///////////////////////////////////////////////////////////////////////////////////////////////////////////////////
	ELSIF StartAction('Nom Action') THEN
		CASE G_Match.iEtapeAction OF
			0:
				IF "CONDITION POUR L'ETAPE SUIVANTE" THEN
					Next(); //etape suivante
				END_IF
			1:
				IF "FIN DE L'ACTION" THEN
					FinishAction(0,0);
				END_IF
		END_CASE
____________________________________________________________________________________________________________________

-> CASE POUR UNE ACTION ASYNCHRONE AVEC LE TABLEAU 
continue la suite du Tableau et l'action en même temps. Si le tableau arrive à une autre action, 
l'action asynchrone est terminée avant de commencer la prochaine action

///////////////////////////////////////////////////////////////////////////////////////////////////////////////////
	ELSIF StartAction('Nom Action') THEN
		CASE G_Match.iEtapeAction OF
			0:
				G_Match.iEtapeAction := G_Match.iEtapeAction + 1;
			1:
				FinishAction(StartAsync := TRUE,0);
			2:
				FinishAction(0,StopAsync := TRUE);
		END_CASE
____________________________________________________________________________________________________________________
*)
END_ACTION

ACTION _5_Interruption_active:
ITMotion.odometrie.M_reset_moteurs();

//Si le robot est bloqué depuis trop longtemps, il essaye différentes actions
IF IbAbortTask THEN
	//Check si c'est possible de reculer en attendant
	(*
	G_Odometrie.lrPositionX;
	G_Odometrie.lrPositionY;
	G_Match.Tableau[G_Match.iLigne].lrPositionX_mm;
	G_Match.Tableau[G_Match.iLigne].lrPositionY_mm;
	G_Balise.lrCoord_X1;
	G_Balise.lrCoord_Y1;
	G_Balise.lrDistance_1;
	*)

	//Sinon calcule les points de la mission en cours
	
	//Vérifie les stratégie possible selon la position
	
	//Choisi la meilleur stratégie à adopter
	
	//modifie le tableau
	
	pass();
END_IF

(*
Adaptation de la stratégie:
- Calcul des points restants
- Recherche de la prochaine stratégie
- Adaptation potentiel du programme
- Changement d'étape et déduction de points
*)

(*
- Tourner 90 degré
- move curve
- reprise de trajectoire

if coordX < 0 or coordX > 3000 or coordY > 2000 or coordY < 0 then
*)
END_ACTION

ACTION _6_Timeout_active:
//S'il ne reste plus de temps pour le match, le robot entamme la manoeuvre pour rentrer à la base
tempTableau.TypeTache := eChangementTache;
tempTableau.EtapeCible := 'retour base';
ReplaceStep(tempTableau);
G_Match.RetourEnCours := TRUE;
END_ACTION

ACTION _7_EndMatch_active:

VisuElems.CURRENTVISU 	:= 'V_Fin_Match';

//arrêt de tous les mouvements
IF G_Match.MatchEnCours THEN
	FOR G_EndMatch.icounter := 1 TO IiNumDynamixel DO
		ITAction.DXLIN[G_EndMatch.icounter].bGetLoad 		:= FALSE;
		ITAction.DXLIN[G_EndMatch.icounter].bGetMovement 	:= FALSE;
		ITAction.DXLIN[G_EndMatch.icounter].bGetPosition 	:= FALSE;

		ITAction.DXLIN[G_EndMatch.icounter].ParamReset_BOOL := TRUE;
		ITAction.DXLIN[G_EndMatch.icounter].bStopPosition 	:= TRUE;
	END_FOR
	
	QbMoteurStop 			:= TRUE;
	G_Match.MatchEnCours 	:= FALSE;
	G_Match.RetourEnCours	:= FALSE;
	baseTime := TIME();
END_IF

//attente pour être sûr que tout soit bien arrêté
IF delay(baseTime, T#0.5S)THEN
	QbMoteurStop 			:= FALSE;
	QbstartBalise 			:= FALSE;
	QbmoteurPower 			:= FALSE;
	
	FOR G_EndMatch.icounter := 1 TO IiNumDynamixel DO
		IF ITAction.DXLOUT[G_EndMatch.icounter].bStopPosition THEN 
			ITAction.DXLIN[G_EndMatch.icounter].bStopPosition := FALSE;
		END_IF
	END_FOR
	
	IF NOT IbStartMatch THEN
			G_EndMatch.bShutdown_done := TRUE;
	END_IF
END_IF;
END_ACTION

ACTION _Config_Visu_active:
IF G_Visus.bConfigEnable THEN 
	VisuElems.CURRENTVISU := 'V_Config';
	//Move robot
	ITMotion.odometrie.M_move_to_coordonne(
	x 			:= G_Visus.lrConfigPosX,
	y 			:= G_Visus.lrConfigPosY,
	lrSpeed 	:= G_Visus.lrConfigVitesse,
	bExecute 	:= G_Visus.bConfigStart,
	bbackward	:= G_Visus.bConfigMarcheArriere,
	bDone 		=> G_Visus.bConfigMoveDone);
	
	//set acceleration / deceleration
	IF G_Visus.lrConfigAcc <> 0 OR G_Visus.lrConfigDecc <> 0 THEN
		ITMotion.odometrie.M_set_acceleration(lrAcc := G_Visus.lrConfigAcc, lrDecc := G_Visus.lrConfigDecc);
	END_IF
	
	//balise on
	QbstartBalise := G_Visus.bConfigBalise;
	
	//moteur on
	QbmoteurPower := G_Visus.bConfigMoteurPower;
	
	//bouton reset
	IF G_Visus.bConfigReset THEN 
		ITMotion.odometrie.M_init_coordonne(bChoixCote := G_Visus.bConfigChoixCote);
	END_IF
	
	//erreur et pourcentage 
	G_Visus.lrConfigErreurX := ABS(G_odometrie.lrPositionX - G_Visus.lrConfigPosX);
	G_Visus.lrConfigErreurY := ABS(G_odometrie.lrPositionY - G_Visus.lrConfigPosY);
	G_Visus.lrConfigErreurX_Pourcent := ABS(G_Visus.lrConfigErreurX/G_odometrie.lrPositionX)*100;
	G_Visus.lrConfigErreurY_Pourcent := ABS(G_Visus.lrConfigErreurY/G_odometrie.lrPositionY)*100;

ELSE// désactivation du mode config
	
	//remise à 0 des valeurs
	QbstartBalise := FALSE;	
	QbmoteurPower := FALSE;
	G_Visus.lrConfigErreurX :=0 ;
	G_Visus.lrConfigErreurY := 0;
	G_Visus.lrConfigErreurX_Pourcent := 0;
	G_Visus.lrConfigErreurY_Pourcent := 0;
	G_Visus.bConfigStart := 0;
	
	//retour au menu
	VisuElems.CURRENTVISU := 'V_Menu';
END_IF

//On doit refaire un init après être sorti du mode config
G_init.binitDone := FALSE;

//mouvement prêt à être effectué
G_Visus.bConfigMoteurReady := IbMoteurOn;

//Indicateur pour dire que le robot est prêt à effectuer un déplacement
IF G_Visus.bConfigMoveDone THEN 
	G_Visus.bConfigStart := FALSE;
END_IF

IF G_Visus.bConfigMoteurReady AND (G_Visus.bConfigStart AND G_Visus.bConfigMoveDone OR NOT G_Visus.bConfigStart)THEN 
	G_Visus.bConfigReady := TRUE;
ELSE
	G_Visus.bConfigReady := FALSE;	
END_IF
END_ACTION

ACTION _Test_Visu_active:
//quitte le mode visu si on retourne au menu
IF VisuElems.CURRENTVISU = 'V_Test' THEN
	G_Visus.bTestEnable := TRUE;
ELSE
	G_Visus.bTestEnable := FALSE;
END_IF

//On doit refaire un init après être sorti du mode Test
G_init.binitDone := FALSE;

IF G_Visus.bTestEnable THEN 
	IF    G_Visus.sTestBouton1 THEN
		G_Match.Tableau[G_Match.iLigne].TypeAction := G_Visus.sTestFunction1;
	ELSIF G_Visus.sTestBouton2 THEN
		G_Match.Tableau[G_Match.iLigne].TypeAction := G_Visus.sTestFunction2;
	ELSIF G_Visus.sTestBouton3 THEN
		G_Match.Tableau[G_Match.iLigne].TypeAction := G_Visus.sTestFunction3;
	ELSIF G_Visus.sTestBouton4 THEN
		G_Match.Tableau[G_Match.iLigne].TypeAction := G_Visus.sTestFunction4;
	ELSIF G_Visus.sTestBouton5 THEN
		G_Match.Tableau[G_Match.iLigne].TypeAction := G_Visus.sTestFunction5;
	ELSIF G_Visus.sTestBouton6 THEN
		G_Match.Tableau[G_Match.iLigne].TypeAction := G_Visus.sTestFunction6;
	END_IF
	
	// TO DO !!!
	//Définir le nom des actions testées 
	G_Visus.sTestFunction1 := 'Dynamixel position 4095';
	G_Visus.sTestFunction2 := 'Dynamixel position 0';
	G_Visus.sTestFunction3 := 'None';
	G_Visus.sTestFunction4 := 'None';
	G_Visus.sTestFunction5 := 'None';
	G_Visus.sTestFunction6 := 'None';
	
	///////////////////////////////////////////////////////////////////////////////////////////////////////////////////
	// GESTION DES ACTIONS 
	///////////////////////////////////////////////////////////////////////////////////////////////////////////////////
	IF StartAction('Dynamixel position 4095') THEN
		CASE G_Match.iEtapeAction OF
			0:
				ITAction.DXLIN[ITAction.MoteurXL1].bPosition := TRUE;
				ITAction.DXLIN[ITAction.MoteurXL1].ParamPosition_DINT := 4095;
				ITAction.DXLIN[ITAction.MoteurXL1].ParamSpeed_INT := 500;
				IF ITAction.DXLOUT[ITAction.MoteurXL1].bPosition THEN
					ITAction.DXLIN[ITAction.MoteurXL1].bPosition := FALSE;
					Next();
				END_IF
			1:
				ITAction.DXLIN[ITAction.MoteurXL1].bGetPosition := TRUE;
				IF PlusOuMoins(ITAction.DXLOUT[ITAction.MoteurXL1].INFO_Position_dint, 4095, 15) THEN 
					ITAction.DXLIN[ITAction.MoteurXL1].bGetPosition := FALSE;
					FinishAction(0);
				END_IF
		END_CASE
	//__________________________________________________________________________________________________________________
	///////////////////////////////////////////////////////////////////////////////////////////////////////////////////			
	ELSIF StartAction('Dynamixel position 0') THEN
		CASE G_Match.iEtapeAction OF
			0:
				ITAction.DXLIN[ITAction.MoteurXL1].bPosition := TRUE;
				ITAction.DXLIN[ITAction.MoteurXL1].ParamPosition_DINT := 1;
				ITAction.DXLIN[ITAction.MoteurXL1].ParamSpeed_INT := 1030;
				IF ITAction.DXLOUT[ITAction.MoteurXL1].bPosition THEN
					ITAction.DXLIN[ITAction.MoteurXL1].bPosition := FALSE;
					Next();;
				END_IF
			1:
				ITAction.DXLIN[ITAction.MoteurXL1].bGetPosition := TRUE;
				IF PlusOuMoins(ITAction.DXLOUT[ITAction.MoteurXL1].INFO_Position_dint, 1, 15) THEN 
					ITAction.DXLIN[ITAction.MoteurXL1].bGetPosition := FALSE;
					FinishAction(0);
				END_IF
		END_CASE
	//__________________________________________________________________________________________________________________
	///////////////////////////////////////////////////////////////////////////////////////////////////////////////////	
	END_IF
	
	//Action terminée
	if G_Match.bActionFinie then
		G_Match.Tableau[G_Match.iLigne].TypeAction := '';
		G_Match.bActionFinie := FALSE;
		G_Match.iEtapeAction := 0;
		
		G_Visus.sTestBouton1 := FALSE;
		G_Visus.sTestBouton2 := FALSE;
		G_Visus.sTestBouton3 := FALSE;
		G_Visus.sTestBouton4 := FALSE;
		G_Visus.sTestBouton5 := FALSE;
		G_Visus.sTestBouton6 := FALSE;
	END_IF

ELSE// désactivation du mode Test
	//remise à 0 des valeurs
	G_Match.bActionFinie := FALSE;
	G_Match.Tableau[G_Match.iLigne].TypeAction := '';
	G_Match.iEtapeAction := 0;
	
	G_Visus.sTestBouton1 := FALSE;
	G_Visus.sTestBouton2 := FALSE;
	G_Visus.sTestBouton3 := FALSE;
	G_Visus.sTestBouton4 := FALSE;
	G_Visus.sTestBouton5 := FALSE;
	G_Visus.sTestBouton6 := FALSE;
	
	FOR G_Match.icounter := 1 TO IiNumDynamixel DO
		ITAction.DXLIN[G_Match.icounter].bGetLoad 		:= FALSE;
		ITAction.DXLIN[G_Match.icounter].bGetMovement 	:= FALSE;
		ITAction.DXLIN[G_Match.icounter].bGetPosition 	:= FALSE;
	END_FOR
END_IF
END_ACTION

TRANSITION T_ArreteTout:
IbEndMatch or G_Match.TimeMatch >= T#100s
END_TRANSITION

TRANSITION T_finMatchNormal:
G_Match.Tableau[G_Match.iLigne].TypeTache = eFinParcours;
END_TRANSITION

TRANSITION T_RetourMatch:
NOT IbPauseMotion
END_TRANSITION

TRANSITION T_Timeout:
G_Match.TimeMatch > T#20s and not G_Match.RetourEnCours
END_TRANSITION

END_PROGRAM

// ---- POUs/Action/ITAction.TcPOU
PROGRAM ITAction
(*IMPORTANT !!! à modifier correctment selon les besoins*)
VAR CONSTANT
	//nombre total de dynamixel
	iNombreDynamixel 	: INT := 4;
	iNombreXL			: INT := 2;
	iNombreAX			: INT := 2;
	
	//définition de l'ID des dynamixels, tous les ID doivent se suivrent => ex: moteur_1 := 1,moteur_2 := 2, moteur_3 := 3, etc...
	//Si des moteurs AX-12A sont présents, leur ID doivent aller après celles des moteurs XL430 ou XL330 => ex: XL430_moteur_5 := 5, AX12A_moteur_1 := 6, etc...
	MoteurXL1 			: INT := 1; //exemple XL430
	MoteurXL2			: INT := 2;
	MoteurAX1 			: INT := 3; //exemple AX12A
	MoteurAX2			: INT := 4;
END_VAR	

VAR_INPUT
	//démarrage et arrêt du script python
	IbStartPyscript 	: BOOL;
	IbStopPyscript		: BOOL;

	//envoi de commande aux moteurs Dynamixel
	DXLIN 				: ARRAY [1..iNombreDynamixel] OF ST_Dynamixel_Control_Input;
END_VAR

VAR_OUTPUT
	QbPyScriptRunning 	: BOOL; //le script python est actif
	QiNombreDynamixel	: INT;
	//retour d'informations des moteurs Dynamixel
	DXLOUT 				: ARRAY [1..iNombreDynamixel] OF ST_Dynamixel_Control_Output;
END_VAR

QiNombreDynamixel := iNombreDynamixel;
P_DXL_launch_pyscript(bstart := IbStartPyscript, bstop := IbStopPyscript);
QbPyScriptRunning := P_DXL_launch_pyscript.bActive;
P_connect_DXL(DXL_IN := DXLIN, DXL_OUT := DXLOUT);

END_PROGRAM

// ---- POUs/Action/Dynamixel/P_DXL_launch_pyscript.TcPOU
PROGRAM P_DXL_launch_pyscript
VAR_INPUT 
	bstart : BOOL;
	bstop : BOOL;
END_VAR
VAR_OUTPUT
	bActive : BOOL;
END_VAR
VAR
	start_python		:NT_StartProcess;
	get_AMSNETID		:FB_GetLocalAmsNetId;
	sPath 				:STRING:= '/C Python Dev\DXL_LIB\';
	sPython_script 		:STRING:= 'DXL_PYADS_PORT.py';
	sAMSNETID 			:STRING;	
	sLaunchCommandLine 	:STRING;
	bBusy				:BOOL;
	
	bRestart_active : BOOL;
END_VAR

//AMSnetID de l'automate
get_AMSNETID(bExecute:=TRUE,AddrString=>sAMSNETID, bBusy=>bBusy);

//ligne de commande dans le terminal pour lancer le script python
sLaunchCommandLine := CONCAT(sPath, sPython_script);
sLaunchCommandLine := CONCAT(sLaunchCommandLine, ' -a ');
sLaunchCommandLine := CONCAT(sLaunchCommandLine, sAMSNETID);

//lance une commande dans le terminal windows pour lancer le script python
//la commande est lancée depuis C:\Windows\SysWOW64\
IF NOT bBusy THEN
	start_python(
	NETID:= '',
	PATHSTR:= 'C:\Windows\System32\cmd.exe',
	DIRNAME:= '',
	COMNDLINE:= sLaunchCommandLine,
	START:= G_DXL.bRestart_py_script,
	TMOUT := T#5S,
	Busy=>,
	ERR=> ,
	ERRID=>); 
END_IF


IF bstart OR bRestart_active THEN 
	// active le script python 1 fois (done_internal bloque la réactivation une fois qu'il a été effectué)
	IF NOT G_DXL.bRestart_py_script AND NOT bRestart_active THEN
		G_DXL.bRestart_py_script := TRUE;
		bRestart_active := TRUE;
	END_IF
	
	// désactive le script python si il était activé
	IF G_DXL.bRestart_py_script AND NOT G_DXL.bPyscript_running AND NOT bRestart_active THEN
		G_DXL.bRestart_py_script := FALSE;	
	END_IF
	
	// libére la réactivation du script python lorsqu'il à redémarré
	IF bRestart_active AND G_DXL.bPyscript_running THEN
		bRestart_active := FALSE;
	END_IF
END_IF

//arrête le script python
IF bStop THEN 
	G_DXL.bStop_python_script := TRUE;
ELSE
	G_DXL.bStop_python_script := FALSE;
END_IF

bActive := G_DXL.bPyscript_running;

END_PROGRAM

// ---- POUs/Action/Dynamixel/P_Connect_DXL.TcPOU
PROGRAM P_Connect_DXL
VAR_IN_OUT
	DXL_IN 	: ARRAY [1..ITAction.iNombreDynamixel] OF ST_Dynamixel_Control_Input;
	DXL_OUT : ARRAY [1..ITAction.iNombreDynamixel] OF ST_Dynamixel_Control_Output;
END_VAR
VAR
	icounter : INT;
END_VAR

FOR icounter := 1 TO ITAction.iNombreDynamixel DO
	IF icounter <= ITAction.iNombreXL THEN //Définition des moteurs XL430 et XL330
		DXL_IN[icounter].TypeXL							(id:= icounter);
		DXL_IN[icounter].TypeXL.send_enable_torque		(EN:=DXL_IN[icounter].bEnableTorque, 	done=> DXL_OUT[icounter].bEnableTorque);
		DXL_IN[icounter].TypeXL.send_disable_torque		(EN:=DXL_IN[icounter].bDisableTorque, 	done=> DXL_OUT[icounter].bDisableTorque);
		DXL_IN[icounter].TypeXL.send_led_on				(EN:=DXL_IN[icounter].bLedOn, 			done=> DXL_OUT[icounter].bLedOn);		
		DXL_IN[icounter].TypeXL.send_led_off			(EN:=DXL_IN[icounter].IbLedOff, 		done=> DXL_OUT[icounter].bLedOff);
		DXL_IN[icounter].TypeXL.send_operating_mode		(EN:=DXL_IN[icounter].bOperatingMode,	done=> DXL_OUT[icounter].bOperatingMode,mode:= DXL_IN[icounter].ParamOperatingMode_string);
		DXL_IN[icounter].TypeXL.send_position			(EN:=DXL_IN[icounter].bPosition, 		done=> DXL_OUT[icounter].bPosition, position 	:= DXL_IN[icounter].ParamPosition_DINT, vitesse:= DXL_IN[icounter].ParamSpeed_INT);
		DXL_IN[icounter].TypeXL.send_stop_position		(EN:=DXL_IN[icounter].bStopPosition, 	done=> DXL_OUT[icounter].bStopPosition,reset:= DXL_IN[icounter].ParamReset_BOOL);
		DXL_IN[icounter].TypeXL.send_reset_position		(EN:=DXL_IN[icounter].bResetPosition, 	done=> DXL_OUT[icounter].bResetPosition);
		DXL_IN[icounter].TypeXL.send_acceleration		(EN:=DXL_IN[icounter].bAcceleration,	done=> DXL_OUT[icounter].bAcceleration, acceleration:= DXL_IN[icounter].ParamAcceleration_USINT, speed:=DXL_IN[icounter].ParamSpeed_INT);
		DXL_IN[icounter].TypeXL.send_velocity			(EN:=DXL_IN[icounter].bVelocity, 		done=> DXL_OUT[icounter].bVelocity, vitesse := DXL_IN[icounter].ParamSpeed_INT);
	    DXL_IN[icounter].TypeXL.get_load				(EN:=DXL_IN[icounter].bGetLoad, 		load=> DXL_OUT[icounter].INFO_load_int);
		DXL_IN[icounter].TypeXL.get_movement			(EN:=DXL_IN[icounter].bGetMovement, 	mouvement=> DXL_OUT[icounter].INFO_Mouvement_bool);
		DXL_IN[icounter].TypeXL.get_position			(EN:=DXL_IN[icounter].bGetPosition,	position=> DXL_OUT[icounter].INFO_Position_dint);
	ELSIF icounter > ITAction.iNombreAX THEN //définition des moteurs AX-12A
		DXL_IN[icounter].TypeAX							(id:= icounter);
		DXL_IN[icounter].TypeAX.send_enable_torque		(EN:=DXL_IN[icounter].bEnableTorque, 	done=> DXL_OUT[icounter].bEnableTorque);
		DXL_IN[icounter].TypeAX.send_disable_torque		(EN:=DXL_IN[icounter].bDisableTorque, 	done=> DXL_OUT[icounter].bDisableTorque);
		DXL_IN[icounter].TypeAX.send_led_on				(EN:=DXL_IN[icounter].bLedOn, 			done=> DXL_OUT[icounter].bLedOn);		
		DXL_IN[icounter].TypeAX.send_led_off			(EN:=DXL_IN[icounter].IbLedOff, 		done=> DXL_OUT[icounter].bLedOff);
		DXL_IN[icounter].TypeAX.send_operating_mode		(EN:=DXL_IN[icounter].bOperatingMode,	done=> DXL_OUT[icounter].bOperatingMode, mode:=DXL_IN[icounter].ParamOperatingMode_string, );
		DXL_IN[icounter].TypeAX.send_position			(EN:=DXL_IN[icounter].bPosition, 		done=> DXL_OUT[icounter].bPosition, position := DXL_IN[icounter].ParamPosition_DINT, vitesse:=DXL_IN[icounter].ParamSpeed_INT);
		DXL_IN[icounter].TypeAX.send_stop_position		(EN:=DXL_IN[icounter].bStopPosition, 	done=> DXL_OUT[icounter].bStopPosition);
		DXL_IN[icounter].TypeAX.send_velocity			(EN:=DXL_IN[icounter].bVelocity, 		done=> DXL_OUT[icounter].bVelocity, vitesse := DXL_IN[icounter].ParamSpeed_INT);
		DXL_IN[icounter].TypeAX.get_load				(EN:=DXL_IN[icounter].bGetLoad, 		load=> DXL_OUT[icounter].INFO_load_int);
		DXL_IN[icounter].TypeAX.get_movement			(EN:=DXL_IN[icounter].bGetMovement, 	mouvement=> DXL_OUT[icounter].INFO_Mouvement_bool);
		DXL_IN[icounter].TypeAX.get_position			(EN:=DXL_IN[icounter].bGetPosition,	position=> DXL_OUT[icounter].INFO_Position_dint);
	END_IF
END_FOR

END_PROGRAM

// ---- POUs/Utillity/Structure/Action/FinishAction.TcPOU
FUNCTION FinishAction 
VAR_INPUT
	StartAsync : BOOL := FALSE;
END_VAR
VAR
END_VAR

G_Match.bActionFinie := TRUE; //arrête l'action sans arrêter la partie asynchrone
IF NOT StartAsync THEN        //arrête l'action asynchrone
	G_Match.iAsyncAction := ''; 
	G_Match.iEtapeAction := 0;
END_IF

END_FUNCTION

// ---- POUs/Structure/Actions/F_DXL_Position.TcPOU
FUNCTION F_DXL_Position : bool
VAR_INPUT
	position:DINT;
	speed	:INT;
	ID		:INT;
END_VAR

CASE G_Match.iEtapeAction OF
	0:
		ITAction.DXLIN[ID].bPosition := TRUE;
		ITAction.DXLIN[ID].ParamPosition_DINT := position;
		ITAction.DXLIN[ID].ParamSpeed_INT := speed;
		IF ITAction.DXLOUT[ID].bPosition THEN
			ITAction.DXLIN[ID].bPosition := FALSE;
			FinishAction(1);
			Next();;
		END_IF
	1:
		ITAction.DXLIN[ID].bGetPosition := TRUE;
		IF PlusOuMoins(ITAction.DXLOUT[ID].INFO_Position_dint, 0, 15) THEN 
			ITAction.DXLIN[ITAction.MoteurXL1].bGetPosition := FALSE;
			FinishAction(0);
		END_IF
END_CASE

END_FUNCTION

// ---- POUs/Structure/Actions/F_DXL_Reset.TcPOU
FUNCTION F_DXL_Reset : bool
VAR_INPUT
	ID:INT;
	offset:DINT;
	
END_VAR
VAR_IN_OUT
	baseTime:TIME;
END_VAR
VAR
END_VAR

CASE G_Match.iEtapeAction OF
	0:
		ITAction.DXLIN[ID].ParamPosition_DINT := 100000;
		ITAction.DXLIN[ID].ParamSpeed_INT := 100;
		
		ITAction.DXLIN[ID].bPosition := TRUE;
		IF ITAction.DXLOUT[ID].bPosition THEN
			ITAction.DXLIN[ID].bPosition := FALSE;
			baseTime := TIME();
			Next();
		END_IF
	1:
		IF delay(baseTime,T#1S)THEN
			next();
		END_IF;
	2:
		G_Visus.bMatchEnemi := TRUE;
		ITAction.DXLIN[ID].bGetLoad := TRUE;
		IF  G_IO.bCaptDepart OR ITAction.DXLOUT[ID].INFO_load_int >= 150 THEN
			ITAction.DXLIN[ITAction.MoteurXL2].bGetLoad := FALSE;
			next();
		END_IF
	3:
		G_Visus.bMatchEnemi := FALSE;
		ITAction.DXLIN[ID].ParamReset_BOOL := TRUE;
		ITAction.DXLIN[ID].bStopPosition := TRUE;
		IF ITAction.DXLOUT[ID].bStopPosition THEN 
			ITAction.DXLIN[ID].bStopPosition := FALSE;
			next();
		END_IF
	4:
		ITAction.DXLIN[ID].bPosition := TRUE;
		ITAction.DXLIN[ID].ParamPosition_DINT := offset;
		ITAction.DXLIN[ID].ParamSpeed_INT := 500;
		IF ITAction.DXLOUT[ID].bPosition THEN
			ITAction.DXLIN[ID].bPosition := FALSE;
			FinishAction(0);
		END_IF
END_CASE

END_FUNCTION

// ---- POUs/Utillity/Structure/Tableau/ReplaceStep.TcPOU
FUNCTION ReplaceStep : bool
VAR_INPUT
	step:ST_Tableau;
END_VAR
VAR
END_VAR

//change l'étape actuelle
G_Match.Tableau[G_Match.iLigne] := step;

END_FUNCTION

// ---- POUs/Communication/ITCommunication.TcPOU
PROGRAM ITCommunication
VAR_INPUT
	IbStartConnection:BOOL;
	IbPublishStart:BOOL;
END_VAR
VAR_OUTPUT
	QbOnline : BOOL;
END_VAR
VAR
	//Lit l'adresse IP de l'automate
	FB_MDP_NIC_Read    : FB_MDP_NIC_Read;
	iAddPoint		   : INT;
END_VAR

FB_MDP_NIC_Read(bExecute := True, tTimeout := DEFAULT_ADS_TIMEOUT);
MQTT(IsHostIP := FB_MDP_NIC_Read.stMDP_ModuleContent.sIPAddress, IbConnect := IbStartConnection, IsTopicOut := 'StartPamis', IsTopicIn := 'FinParcours', IbPublishStart := IbPublishStart, IsPayload := 'Start', QiAddPoint := iAddPoint);
QbOnline := MQTT.QbOnline;

END_PROGRAM

// ---- POUs/Communication/MQTT.TcPOU
PROGRAM MQTT
VAR_INPUT
	IsHostIP 	: STRING;					//Adresse IP du broker Mosquitto qui tourne sur la partie windows de la PLC
	IbConnect 	: BOOL;						//Commence la connection MQTT
	
	IsTopicOut 	: STRING;					//Nom du Topic où la PLC publie des chose
	IsTopicIn 	: STRING;					//Nom du Topic où la PLC est souscrite (lis les informations)
	IbPublishStart : BOOL;					//Un front montant publie le message IsPayload dans le topic IsTopicOut
	IsPayload : STRING;						//Message à publier dans le topic
	
END_VAR
VAR_OUTPUT
	QbOnline : BOOL;						//Communication MQTT en ligne
END_VAR
VAR_IN_OUT
	QiAddPoint : INT;						//Donne l'ordre d'ajouter des points	
END_VAR
VAR
fbMqttClient 	: FB_IotMqttClient;			//FB de gestion de la communication MQTT
fbMessageQueue 	: FB_IotMqttMessageQueue;	//Zone tampon de stockage des messages reçus
fbMessage 		: FB_IotMqttMessage;		//Formattage des message MQTT reçu

RT_Publish 		: R_TRIG;					//Front montant pour la publication

bSubscribed : BOOL;							//Souscription au topic effectué

{attribute 'TcEncoding':='UTF-8'}
sPayloadRcv 	: STRING(255);				//Contenu du message souscrit (valeur reçue)
iNumPamiDone	: INT;						//Numéro du PAMI qui à fini son action
END_VAR

IF _TaskInfo[GETCURTASKINDEXEX()].FirstCycle THEN	//Lancement de la recherche de broker
	fbMqttClient.sHostName 		:= IsHostIP;		//Adresse IP d'ou se situe le broker (donc sur un Raspberry dans Node-red)
	fbMqttClient.nHostPort 		:= 1883;			//Port de communication du broker
	fbMqttClient.sClientId 		:= 'Bobst PLC';
	fbMqttClient.sTopicPrefix 	:= '';
	fbMqttClient.nKeepAlive 	:= 10;
	fbMqttClient.ipMessageQueue := fbMessageQueue;	//Sert à stocker les messages souscrit avant de les traiter
END_IF

//Lancement de la connexion MQTT
fbMqttClient.Execute(IbConnect);	
QbOnline := fbMqttClient.bConnected AND bSubscribed;

//Si on est connecté au broker alors...
IF fbMqttClient.bConnected THEN	

	//*** Souscrire à un topic ***//
	IF NOT bSubscribed THEN		//Signal pour lancer la souscription à un message
		bSubscribed := fbMqttClient.Subscribe(sTopic:=IsTopicIn,  eQoS:=TcIotMqttQos.AtMostOnceDelivery);
	END_IF
	
	//*** Publier un message ***//
	RT_Publish(clk:=IbPublishStart);
	IF  RT_Publish.Q THEN //Lorsque ce signal est à 1, on publie un message
		fbMqttClient.Publish( sTopic  		:= IsTopicOut,	//On écrit le nom du Topic d'un message à envoyer
							  pPayload		:= ADR(IsPayload),	//On écrit le contenu du message à envoyer (valeur à envoyer)
							  nPayloadSize	:= SIZEOF(IsPayload),	//On indique la taille du STRING donc le nombre de caractère.
							  eQoS			:= TcIotMqttQos.AtMostOnceDelivery,	//Qualité de service, à laisser comme cela
							  bRetain		:= FALSE,	//à laisser comme cela
							  bQueue		:= FALSE );	//à laisser comme cela
	END_IF			
END_IF

//*** Récupérer les messages des topics auquels on est souscris ***//
IF (fbMessageQueue.nQueuedMessages > 0) THEN 
	IF fbMessageQueue.Dequeue(fbMessage:=fbMessage) THEN
		IF fbMessage.CompareTopic(sTopic:=IsTopicIn) THEN
			fbMessage.GetPayload(pPayload:=ADR(sPayloadRcv), nPayloadSize:=SIZEOF(sPayloadRcv), bSetNullTermination:=FALSE);	//Valeur du message 1 reçu
		END_IF
		iNumPamiDone := STRING_TO_INT(RIGHT(sPayloadRcv,1));		
	END_IF
END_IF

//Choisi le nombre de points à ajouter en fonction du message MQTT reçu
CASE iNumPamiDone OF
	0:
		pass();
	1:
		QiAddPoint := 10;
		iNumPamiDone := 0;
	2:
		QiAddPoint := 10;
		iNumPamiDone := 0;
	3:
		QiAddPoint := 10;
		iNumPamiDone := 0;
	4:		
		QiAddPoint := 10;
		iNumPamiDone := 0;
END_CASE

END_PROGRAM

// ---- POUs/Action/Camera OAK-D/FB_CAM.TcPOU
FUNCTION_BLOCK FB_CAM
VAR_INPUT
	bAruco 	: BOOL;
	bProxi	: BOOL;
END_VAR
VAR_OUTPUT
	TAruco 			: ARRAY [0..10] OF INT;
	usiProximite 	: USINT;
END_VAR

//author: Alec Horth

//gestion des fonctionnalités de la caméra
// voir GVL "G_CAM" pour plus de détails d'implémentation
G_CAM.RUN_ARUCO := bAruco;
IF bAruco THEN
	TAruco := G_CAM.tag_aruco;
END_IF

G_CAM.RUN_STEREO := bProxi;
IF bProxi THEN
	usiProximite := G_CAM.proximite;
END_IF

END_FUNCTION_BLOCK

// ---- POUs/Action/Camera OAK-D/P_cam_launch_pyscript.TcPOU
PROGRAM P_cam_launch_pyscript
VAR_INPUT
	bstart 	: BOOL;
	bstop	: BOOL;
END_VAR
VAR_OUTPUT
	bActive	: BOOL;
END_VAR
VAR
	python				:NT_StartProcess;
	get_AMSNETID		:FB_GetLocalAmsNetId;
	path 				:STRING := '/C Python Dev\OAK_D\';
	python_script 		:STRING := 'CAM_PORT.py';
	AMSNETID 			:STRING;
	launchCommandLine 	:STRING(255);
	busy				:BOOL;
	
	bRestartActive		:BOOL;
	bStopActive			:BOOL;
END_VAR

get_AMSNETID(bExecute:=G_CAM.restart_py_script,AddrString=>AMSNETID, bBusy=>busy);

launchCommandLine := CONCAT(path, python_script);
launchCommandLine := CONCAT(launchCommandLine, ' -a ');
launchCommandLine := CONCAT(launchCommandLine, AMSNETID);
if not busy then
	python(
	NETID:= '',
	PATHSTR:= 'C:\Windows\System32\cmd.exe',
	DIRNAME:= '',
	COMNDLINE:= launchCommandLine,
	START:= G_CAM.restart_py_script,
	TMOUT := T#5s,
	BUSY=>,
	ERR=> ,
	ERRID=>);
END_IF

IF bStart AND NOT bRestartActive THEN
	bRestartActive := TRUE;
	G_CAM.restart_py_script:=FALSE;
END_IF
IF bRestartActive AND NOT G_CAM.restart_py_script THEN
	G_CAM.restart_py_script :=TRUE;
END_IF
IF G_CAM.restart_py_script AND NOT bStart THEN 
	bRestartActive := FALSE;
END_IF

IF bStop THEN
	G_CAM.STOP_PYSCRIPT:=TRUE;
END_IF

bActive := G_CAM.bPyscript_running;

END_PROGRAM

// ---- POUs/Action/Dynamixel/FB_DXL_AX12A.TcPOU
FUNCTION_BLOCK FB_DXL_AX12A
VAR_INPUT 
	id : INT; // ID du moteur Dynamixel de 0 à 253. Addresse 254 => broadcast (cible tous les moteurs)
END_VAR
VAR  
	//communication en cours
	com_ongoing : BOOL;
	// modèle du moteur
	motor_type : USINT:= AX12A;
END_VAR
VAR CONSTANT
	//type du moteur
	XL430:USINT:=2;
	AX12A:USINT:=1;
END_VAR

//author: Alec Horth
//mail  : horth.alec@gmail.com

METHOD PROTECTED _end_communication : BOOL
VAR_IN_OUT
	run:BOOL; // arrête la variable qui maintient la fonction en vie 
	started:BOOL; // arrête la variable qui indique que la fonction possède un token
END_VAR
VAR_INST
	pulse : F_TRIG;
	once : bool;
END_VAR
// front descendant activé par le script python et désactivé par la fonction _send()
// confirme que la commande à bien été envoyée
pulse(CLK:=G_DXL.bDone AND started, Q=>);

IF pulse.Q THEN 
	//permet de lancer cette fonction une seule fois, sinon elle relance un cycle de façon involontaire 
	once := TRUE;
END_IF

IF once THEN
	// libère le token
	G_DXL.bToken := G_DXL.iOPEN_TOKEN;
	com_ongoing := FALSE;
	run := FALSE;
	_end_communication := TRUE;
	started := FALSE;
	once := FALSE;
ELSE
	_end_communication := FALSE;
END_IF
END_METHOD

METHOD PROTECTED _send : BOOL
VAR_INPUT
END_VAR
VAR_INST
	once :BOOL; // assure que la commande n'est envoyé qu'une fois
END_VAR
IF G_DXL.bDone THEN 	//confirmation d'acquisition de la commande du script python
	G_DXL.bRun := FALSE; //indique au script python que le message est passé
ELSIF NOT G_DXL.bDone AND NOT once THEN // si la commande n'a pas encore été envoyé, lance la commande
	once := TRUE;
	G_DXL.bRun := TRUE;
END_IF

IF NOT com_ongoing THEN // permet de relancer des commandes lorsque le token est rendu
	once := FALSE;
END_IF
END_METHOD

METHOD PROTECTED _start_communication : BOOL
VAR_IN_OUT
	started:BOOL; //maintient la fonction active tant que le token n'est pas rendu
END_VAR
IF ((G_DXL.bToken = G_DXL.iOPEN_TOKEN OR G_DXL.bToken = id) AND NOT com_ongoing AND NOT G_DXL.bDone) OR started THEN // vérifie que tous les token soient libres
	// attribution du token
	started := TRUE; 
	G_DXL.bToken := id;
	// configure les commandes à envoyer avec le bon ID et le bon type du moteur
	G_DXL.iID := id;
	G_DXL.usiMotor_type := motor_type;
	com_ongoing := TRUE; 
	_start_communication := TRUE;	
ELSE 
	_start_communication := FALSE;
END_IF
END_METHOD

METHOD private BASE_EXEMPLE_FUTUR_MODIF_SEND 
VAR_INPUT
	EN			:BOOL; // un front montant change le taux d'accélération du moteur
	
	//--------------TO DO---------------
	parametre1	:usint;
	parametre2	:INT;
	//----------------------------------

END_VAR
VAR_OUTPUT
	done		:BOOL; //la commande est envoyée, passe à False si EN passe aussi à False
END_VAR
VAR_INST 
	bRun 		:BOOL;
	rtrigPulse 	:R_TRIG;
	bDone_pulse :BOOL;
	bStarted 	:BOOL;
END_VAR
// IL EST POSSIBLE DE MODIFIER LES SECTION "TO DO", LE RESTE NE DOIT PAS ÊTRE MODIFIE

//Activation de la fonction
rtrigPulse(CLK:=EN, Q=>);

IF rtrigPulse.Q THEN
	//Si une autre fonction est déjà en cours de traitement (token déjà pris) cette fonction ne peut pas être effectuée
	//La variable run garde l'ordre d'activation en mémoire et lance la fonction dès que le token est libéré
	bRun := TRUE;
END_IF

IF bRun THEN
	IF _start_communication(started:=bStarted) THEN 	//vérifie si les tokens sont libérés 
		
		//--------------TO DO---------------
		G_DXL.usiFonction := G_DXL.usiGOAL_ACCELERATION; 	// choix de la commande à envoyer		
		G_DXL.usiAcceleration 	:= parametre1;				//paramètre 1
		G_DXL.iSpeed    		:= parametre2;				//paramètre 2 
		//----------------------------------
		
		
		bDone_pulse := _end_communication(run:=bRun, started:=bStarted) AND EN;	//libère le token une fois que la commande est lancée
		_send();																//Envoi de la commande au moteur
	END_IF
END_IF;

IF bDone_pulse AND EN THEN														//Affiche le status d'excution de la fonction
	done := EN;																	//tant que EN est à True
ELSIF bDone_pulse AND NOT EN THEN
	bDone_pulse := FALSE;
END_IF
END_METHOD

METHOD get_load : BOOL
VAR_INPUT
	EN:BOOL; 	// ouvre un canal de transmission avec le moteur 
END_VAR
VAR_OUTPUT
	load:INT; 	// le moteur renvoie le torque qu'il emet à travers le canal (voir dans la méthode pour + d'infos)
				//(AX12A) 0-1023 torque est dans le sens inverse des aiguilles d'une montre, entre 1024 et 2047 le torque est dans le sens des aiguilles d'une montre
				//(XL430) +- 1000 pour mille du torque maximum si la valeur est positive => le torque est dans le sens inverse des aiguilles d'une montre
END_VAR
VAR_inst 
	run :BOOL;
	pulse : R_TRIG;
	started: BOOL;
END_VAR
//ouvre le canal de transmission
pulse(CLK:=EN, Q=>);

IF pulse.Q THEN
	//Si une autre fonction est déjà en cours de traitement (token déjà pris) le canal ne peut pas être ouvert
	//La variable run garde l'ordre d'activation en mémoire et ouvre le canal dès que le token est libéré
	run := TRUE;
END_IF

IF run THEN 
	IF _start_communication(started := started) THEN 	// Vérifie si le token est libre
		G_DXL.usiFonction := G_DXL.usiGET_PRESENT_LOAD;	// configure le canal à ouvrir
		G_DXL.bRun := TRUE;								// envoie la commande au script python
		load := G_DXL.iDxl_load;						// si le canal est ouvert, renvoie la valeur actuelle du torque émit pas le moteur
	END_IF
	IF NOT EN THEN
		G_DXL.bRun 	:= FALSE;						    //ferme le canal
		G_DXL.iDxl_load := -9000;						//remet une valeur par défault
		_end_communication(run:=run,started := started);//libère le token
	END_IF;
ELSE
	load := -9000;										//valeur par défaut
END_IF
END_METHOD

METHOD get_movement : BOOL
VAR_INPUT
	EN:BOOL; 	// ouvre un canal de transmission avec le moteur 
END_VAR
VAR_OUTPUT
	mouvement:BOOL; // le moteur renvoie si il est en mouvement(TRUE) ou non (FALSE)
END_VAR
VAR_INST 
	run :BOOL;
	pulse : R_TRIG;
	started: BOOL;
END_VAR
//ouvre le canal de transmission
pulse(CLK:=EN, Q=>);

IF pulse.Q THEN
	//Si une autre fonction est déjà en cours de traitement (token déjà pris) le canal ne peut pas être ouvert
	//La variable run garde l'ordre d'activation en mémoire et ouvre le canal dès que le token est libéré
	run := TRUE;
END_IF

IF run THEN 
	IF _start_communication(started := started) THEN 	// Vérifie si le token est libre
		G_DXL.usiFonction := G_DXL.usiGET_PRESENT_MOVEMENT;	// configure le canal à ouvrir
		G_DXL.bRun := TRUE;								// envoie la commande au script python
		mouvement := G_DXL.bDxl_movement;				// status du mouvement du moteur Dynamixel
	END_IF
	IF NOT EN THEN
		G_DXL.bRun 	:= FALSE;						    //ferme le canal
		G_DXL.bDxl_movement := 1;						//remet une valeur par défault
		_end_communication(run:=run,started := started);//libère le token
	END_IF;
ELSE
	mouvement := 1;										//valeur par défaut
END_IF
END_METHOD

METHOD get_position : BOOL
VAR_INPUT
	EN:BOOL; 	// ouvre un canal de transmission avec le moteur 
END_VAR
VAR_OUTPUT
	position:DINT; //(AX12A sur 300 degrés)0-1023 ou (XL430 sur 360 degrés)0-4095 ou (XL430 en multitours)+- 1'048'575
END_VAR
VAR_INST 
	run :BOOL;
	pulse : R_TRIG;
	started: BOOL;
END_VAR
//ouvre le canal de transmission
pulse(CLK:=EN, Q=>);

IF pulse.Q THEN
	//Si une autre fonction est déjà en cours de traitement (token déjà pris) le canal ne peut pas être ouvert
	//La variable run garde l'ordre d'activation en mémoire et ouvre le canal dès que le token est libéré
	run := TRUE;
END_IF

IF run THEN 
	IF _start_communication(started := started) THEN 	// Vérifie si le token est libre
		G_DXL.usiFonction := G_DXL.usiGET_PRESENT_POSITION;	// configure le canal à ouvrir
		G_DXL.bRun := TRUE;								// envoie la commande au script python
		position := G_DXL.diDxl_position;				//(AX12A sur 300 degrés)0-1023 ou (XL430 sur 360 degrés)0-4095 ou (XL430 en multitours)+- 1'048'575
	END_IF
	IF NOT EN THEN
		G_DXL.bRun 	:= FALSE;						    //ferme le canal
		G_DXL.diDxl_position := -9000;					//remet une valeur par défault
		_end_communication(run:=run,started := started);//libère le token
	END_IF;
ELSE
	position := -9000;									//valeur par défaut
END_IF
END_METHOD

METHOD send_disable_torque 
VAR_INPUT
	EN			:BOOL; // un impulsion active le torque du moteur
END_VAR
VAR_OUTPUT
	done		:BOOL; //la commande est envoyée, passe à False si EN passe aussi à False
END_VAR
VAR_INST 
	run 		:BOOL;
	pulse 		:R_TRIG;
	done_pulse 	:BOOL;
	started 	:BOOL;
END_VAR
//Activation de la fonction
pulse(CLK:=EN, Q=>);

IF pulse.Q THEN
	//Si une autre fonction est déjà en cours de traitement (token déjà pris) cette fonction ne peut pas être effectuée
	//La variable run garde l'ordre d'activation en mémoire et lance la fonction dès que le token est libéré
	run := TRUE;
END_IF

IF run THEN
	IF _start_communication(started:=started) THEN 								//vérifie si les tokens sont libérés 
		G_DXL.usiFonction := G_DXL.usiDISABLE_TORQUE;									//Ecriture de la commande
		done_pulse := _end_communication(run:=run, started:=started) AND EN;	//libère le token une fois que la commande est lancée
		_send();																//Envoi de la commande au moteur
	END_IF
END_IF;

IF done_pulse AND EN THEN														//Affiche le status d'excution de la fonction
	done := EN;																	//tant que EN est à True
ELSIF done_pulse AND NOT EN THEN
	done_pulse := FALSE;
END_IF
END_METHOD

METHOD send_enable_torque 
VAR_INPUT
	EN			:BOOL; // un front montant désactive le torque du moteur 
END_VAR
VAR_OUTPUT
	done		:BOOL; // la commande est envoyée, passe à False si EN passe aussi à False 
END_VAR
VAR_INST 
	run 		:BOOL;
	pulse 		:R_TRIG;
	done_pulse 	:BOOL;
	started 	:BOOL;
END_VAR
//Activation de la fonction
pulse(CLK:=EN, Q=>);

IF pulse.Q THEN
	//Si une autre fonction est déjà en cours de traitement (token déjà pris) cette fonction ne peut pas être effectuée
	//La variable run garde l'ordre d'activation en mémoire et lance la fonction dès que le token est libéré
	run := TRUE;
END_IF

IF run THEN
	IF _start_communication(started:=started) THEN 								//vérifie si les tokens sont libérés 
		G_DXL.usiFonction := G_DXL.usiENABLE_TORQUE;									//Ecriture de la commande
		done_pulse := _end_communication(run:=run, started:=started) AND EN;	//libère le token une fois que la commande est lancée
		_send();																//Envoi de la commande au moteur
	END_IF
END_IF;

IF done_pulse AND EN THEN														//Affiche le status d'excution de la fonction
	done := EN;																	//tant que EN est à True
ELSIF done_pulse AND NOT EN THEN
	done_pulse := FALSE;
END_IF
END_METHOD

METHOD send_led_off 
VAR_INPUT
	EN			:BOOL; // un front montant éteint la LED
END_VAR
VAR_OUTPUT
	done		:BOOL; // la commande est envoyée, passe à False si EN passe aussi à False 
END_VAR
VAR_INST 
	run 		:BOOL;
	pulse 		:R_TRIG;
	done_pulse 	:BOOL;
	started 	:BOOL;
END_VAR
//Activation de la fonction
pulse(CLK:=EN, Q=>);

IF pulse.Q THEN
	//Si une autre fonction est déjà en cours de traitement (token déjà pris) cette fonction ne peut pas être effectuée
	//La variable run garde l'ordre d'activation en mémoire et lance la fonction dès que le token est libéré
	run := TRUE;
END_IF

IF run THEN
	IF _start_communication(started:=started) THEN 								//vérifie si les tokens sont libérés 
		G_DXL.usiFonction := G_DXL.usiLED_OFF;										//Ecriture de la commande
		done_pulse := _end_communication(run:=run, started:=started) AND EN;	//libère le token une fois que la commande est lancée
		_send();																//Envoi de la commande au moteur
	END_IF
END_IF;

IF done_pulse AND EN THEN														//Affiche le status d'excution de la fonction
	done := EN;																	//tant que EN est à True
ELSIF done_pulse AND NOT EN THEN
	done_pulse := FALSE;
END_IF
END_METHOD

METHOD send_led_on 
VAR_INPUT
	EN			:BOOL; // un front montant allume la LED
END_VAR
VAR_OUTPUT
	done		:BOOL; // la commande est envoyée, passe à False si EN passe aussi à False 
END_VAR
VAR_INST 
	run 		:BOOL;
	pulse 		:R_TRIG;
	done_pulse 	:BOOL;
	started 	:BOOL;
END_VAR
//Activation de la fonction
pulse(CLK:=EN, Q=>);

IF pulse.Q THEN
	//Si une autre fonction est déjà en cours de traitement (token déjà pris) cette fonction ne peut pas être effectuée
	//La variable run garde l'ordre d'activation en mémoire et lance la fonction dès que le token est libéré
	run := TRUE;
END_IF

IF run THEN
	IF _start_communication(started:=started) THEN 								//vérifie si les tokens sont libérés 
		G_DXL.usiFonction := G_DXL.usiLED_ON;											//Ecriture de la commande
		done_pulse := _end_communication(run:=run, started:=started) AND EN;	//libère le token une fois que la commande est lancée
		_send();																//Envoi de la commande au moteur
	END_IF
END_IF;

IF done_pulse AND EN THEN														//Affiche le status d'excution de la fonction
	done := EN;																	//tant que EN est à True
ELSIF done_pulse AND NOT EN THEN
	done_pulse := FALSE;
END_IF
END_METHOD

METHOD send_operating_mode 
VAR_INPUT
	EN			:BOOL; // un front montant change le mode de pilotage du moteur
	mode		:STRING;//‘position’ ou 'position_angleMin_angleMax’ => ex: 'position_10_100' ou ‘velocity’

END_VAR
VAR_OUTPUT
	done		:BOOL; //la commande est envoyée, passe à False si EN passe aussi à False 
END_VAR
VAR_INST 
	run 		:BOOL;
	pulse 		:R_TRIG;
	done_pulse 	:BOOL;
	started 	:BOOL;
END_VAR
//Activation de la fonction
pulse(CLK:=EN, Q=>);

IF pulse.Q THEN
	//Si une autre fonction est déjà en cours de traitement (token déjà pris) cette fonction ne peut pas être effectuée
	//La variable run garde l'ordre d'activation en mémoire et lance la fonction dès que le token est libéré
	run := TRUE;
END_IF

IF run THEN
	IF _start_communication(started:=started) THEN 								//vérifie si les tokens sont libérés 
		G_DXL.usiFonction := G_DXL.usiOPERATING_MODE;									//Ecriture de la commande
		G_DXL.sMode := mode;
		done_pulse := _end_communication(run:=run, started:=started) AND EN;	//libère le token une fois que la commande est lancée
		_send();																//Envoi de la commande au moteur
	END_IF
END_IF;

IF done_pulse AND EN THEN														//Affiche le status d'excution de la fonction
	done := EN;																	//tant que EN est à True
ELSIF done_pulse AND NOT EN THEN
	done_pulse := FALSE;
END_IF
END_METHOD

METHOD send_position 
VAR_INPUT
	EN			:BOOL; // un front montant déplace le moteur à la position voulue
	position	:DINT; //(AX12A sur 300 degrés)0-1023 ou (XL430 sur 360 degrés)0-4095 ou (XL430 en multitours)+- 1'048'575
	vitesse		:INT;  //(AX12A)0-1023 ou (XL430)0-1023 
END_VAR
VAR_OUTPUT
	done		:BOOL; // la commande est envoyée, passe à False si EN passe aussi à False 
END_VAR
VAR_INST 
	run 		:BOOL;
	pulse 		:R_TRIG;
	done_pulse 	:BOOL;
	started 	:BOOL;
END_VAR
//Activation de la fonction
pulse(CLK:=EN, Q=>);

IF pulse.Q THEN
	//Si une autre fonction est déjà en cours de traitement (token déjà pris) cette fonction ne peut pas être effectuée
	//La variable run garde l'ordre d'activation en mémoire et lance la fonction dès que le token est libéré
	run := TRUE;
END_IF

IF run THEN
	IF _start_communication(started:=started) THEN 								//vérifie si les tokens sont libérés 
		G_DXL.usiFonction := G_DXL.usiGOAL_POSITION;									//Ecriture de la commande
		G_DXL.diPosition := position;
		G_DXL.iSpeed    := vitesse;
		done_pulse := _end_communication(run:=run, started:=started) AND EN;	//libère le token une fois que la commande est lancée
		_send();																//Envoi de la commande au moteur
	END_IF
END_IF;

IF done_pulse AND EN THEN														//Affiche le status d'excution de la fonction
	done := EN;																	//tant que EN est à True
ELSIF done_pulse AND NOT EN THEN
	done_pulse := FALSE;
END_IF
END_METHOD

METHOD send_stop_position 
VAR_INPUT
	EN			:BOOL; // un front montant arrête le moteur à sa position actuelle
END_VAR
VAR_OUTPUT
	done		:BOOL; // la commande est envoyée, passe à False si EN passe aussi à False 
END_VAR
VAR_INST 
	run 		:BOOL;
	pulse 		:R_TRIG;
	done_pulse 	:BOOL;
	started 	:BOOL;
END_VAR
//Activation de la fonction
pulse(CLK:=EN, Q=>);

IF pulse.Q THEN
	//Si une autre fonction est déjà en cours de traitement (token déjà pris) cette fonction ne peut pas être effectuée
	//La variable run garde l'ordre d'activation en mémoire et lance la fonction dès que le token est libéré
	run := TRUE;
END_IF

IF run THEN
		IF _start_communication(started:=started) THEN 								//vérifie si les tokens sont libérés 
		G_DXL.usiFonction := G_DXL.usiSTOP_POSITION;										//Ecriture de la commande
		done_pulse := _end_communication(run:=run, started:=started) AND EN;		//libère le token une fois que la commande est lancée
		_send();																	//Envoi de la commande au moteur
	END_IF
END_IF;

IF done_pulse AND EN THEN														//Affiche le status d'excution de la fonction
	done := EN;																	//tant que EN est à True
ELSIF done_pulse AND NOT EN THEN
	done_pulse := FALSE;
END_IF
END_METHOD

METHOD send_velocity 
VAR_INPUT
	EN			:BOOL; // un front montant donne une nouvelle vitesse au moteur en mode velocity
	vitesse		:INT;  //(AX12A)0-2047
END_VAR
VAR_OUTPUT
	done		:BOOL; // la commande est envoyée, passe à False si EN passe aussi à False 
END_VAR
VAR_INST 
	run 		:BOOL;
	pulse 		:R_TRIG;
	done_pulse 	:BOOL;
	started 	:BOOL;
END_VAR
//Activation de la fonction
pulse(CLK:=EN, Q=>);

IF pulse.Q THEN
	//Si une autre fonction est déjà en cours de traitement (token déjà pris) cette fonction ne peut pas être effectuée
	//La variable run garde l'ordre d'activation en mémoire et lance la fonction dès que le token est libéré
	run := TRUE;
END_IF

IF run THEN
	IF _start_communication(started:=started) THEN 								//vérifie si les tokens sont libérés 
		G_DXL.usiFonction := G_DXL.usiGOAL_VELOCITY;									//Ecriture de la commande
		G_DXL.iSpeed    := vitesse;
		done_pulse := _end_communication(run:=run, started:=started) AND EN;	//libère le token une fois que la commande est lancée
		_send();																//Envoi de la commande au moteur
	END_IF
END_IF;

IF done_pulse AND EN THEN														//Affiche le status d'excution de la fonction
	done := EN;																	//tant que EN est à True
ELSIF done_pulse AND NOT EN THEN
	done_pulse := FALSE;
END_IF
END_METHOD

END_FUNCTION_BLOCK

// ---- POUs/Action/Dynamixel/FB_DXL_XL.TcPOU
FUNCTION_BLOCK FB_DXL_XL
VAR_INPUT 
	id : INT;
END_VAR
VAR  
	//communication en cours
	com_ongoing	: BOOL;
END_VAR
VAR CONSTANT
	//type du moteur
	XL430:USINT:=2;
	AX12A:USINT:=1;
	
	motor_type : USINT:=XL430;
END_VAR

//author: Alec Horth
//mail  : horth.alec@gmail.com

METHOD PRIVATE _end_communication : BOOL
VAR_IN_OUT
	run:BOOL; // arrête la variable qui maintient la fonction en vie 
	started:BOOL; // arrête la variable qui indique que la fonction possède un token
END_VAR
VAR_INST
	pulse : F_TRIG;
	once : bool;
END_VAR
// front descendant activé par le script python et désactivé par la fonction _send()
// confirme que la commande à bien été envoyée
pulse(CLK:=G_DXL.bDone AND started, Q=>);

IF pulse.Q THEN 
	//permet de lancer cette fonction une seule fois, sinon elle relance un cycle de façon involontaire 
	once := TRUE;
END_IF

IF once THEN
	// libère le token
	G_DXL.bToken := G_DXL.iOPEN_TOKEN;
	com_ongoing := FALSE;
	run := FALSE;
	_end_communication := TRUE;
	started := FALSE;
	once := FALSE;
ELSE
	_end_communication := FALSE;
END_IF
END_METHOD

METHOD PRIVATE _send : BOOL
VAR_INPUT
END_VAR
VAR_INST
	once :BOOL; // assure que la commande n'est envoyé qu'une fois
END_VAR
IF G_DXL.bDone THEN 	//confirmation d'acquisition de la commande du script python
	G_DXL.bRun := FALSE; //indique au script python que le message est passé
ELSIF NOT G_DXL.bDone AND NOT once THEN // si la commande n'a pas encore été envoyé, lance la commande
	once := TRUE;
	G_DXL.bRun := TRUE;
END_IF

IF NOT com_ongoing THEN // permet de relancer des commandes lorsque le token est rendu
	once := FALSE;
END_IF
END_METHOD

METHOD PRIVATE _start_communication : BOOL
VAR_IN_OUT
	started:BOOL; //maintient la fonction active tant que le token n'est pas rendu
END_VAR
IF ((G_DXL.bToken = G_DXL.iOPEN_TOKEN OR G_DXL.bToken = id) AND NOT com_ongoing AND NOT G_DXL.bDone) OR started THEN // vérifie que tous les token soient libres
	// attribution du token
	started := TRUE; 
	G_DXL.bToken := id;
	// configure les commandes à envoyer avec le bon ID et le bon type du moteur
	G_DXL.iID := id;
	G_DXL.usiMotor_type := motor_type;
	com_ongoing := TRUE; 
	_start_communication := TRUE;	
ELSE 
	_start_communication := FALSE;
END_IF
END_METHOD

METHOD private BASE_EXEMPLE_FUTUR_MODIF_SEND : BOOL
VAR_INPUT
	EN			:BOOL; // un front montant change le taux d'accélération du moteur
	
	//--------------TO DO---------------
	parametre1	:usint;
	parametre2	:INT;
	//----------------------------------

END_VAR
VAR_OUTPUT
	done		:BOOL; //la commande est envoyée, passe à False si EN passe aussi à False
END_VAR
VAR_INST 
	bRun 		:BOOL;
	rtrigPulse 	:R_TRIG;
	bDone_pulse :BOOL;
	bStarted 	:BOOL;
END_VAR
// IL EST POSSIBLE DE MODIFIER LES SECTION "TO DO", LE RESTE NE DOIT PAS ÊTRE MODIFIE

//Activation de la fonction
rtrigPulse(CLK:=EN, Q=>);

IF rtrigPulse.Q THEN
	//Si une autre fonction est déjà en cours de traitement (token déjà pris) cette fonction ne peut pas être effectuée
	//La variable run garde l'ordre d'activation en mémoire et lance la fonction dès que le token est libéré
	bRun := TRUE;
END_IF

IF bRun THEN
	IF _start_communication(started:=bStarted) THEN 	//vérifie si les tokens sont libérés 
		
		//--------------TO DO---------------
		G_DXL.usiFonction := G_DXL.usiGOAL_ACCELERATION; 	// choix de la commande à envoyer		
		G_DXL.usiAcceleration 	:= parametre1;				//paramètre 1
		G_DXL.iSpeed    		:= parametre2;				//paramètre 2 
		//----------------------------------
		
		
		bDone_pulse := _end_communication(run:=bRun, started:=bStarted) AND EN;	//libère le token une fois que la commande est lancée
		_send();																//Envoi de la commande au moteur
	END_IF
END_IF;

IF bDone_pulse AND EN THEN														//Affiche le status d'excution de la fonction
	done := EN;																	//tant que EN est à True
ELSIF bDone_pulse AND NOT EN THEN
	bDone_pulse := FALSE;
END_IF
END_METHOD

METHOD get_load 
VAR_INPUT
	EN:BOOL; 	// ouvre un canal de transmission avec le moteur 
END_VAR
VAR_OUTPUT
	load:INT; 	// le moteur renvoie le torque qu'il emet à travers le canal (voir dans la méthode pour + d'infos)
				//(AX12A) 0-1023 torque est dans le sens inverse des aiguilles d'une montre, entre 1024 et 2047 le torque est dans le sens des aiguilles d'une montre
				//(XL430) +- 1000 pour mille du torque maximum si la valeur est positive => le torque est dans le sens inverse des aiguilles d'une montre
	done:bool;
END_VAR
VAR_inst 
	run :BOOL;
	pulse : R_TRIG;
	started: BOOL;
END_VAR
//ouvre le canal de transmission
pulse(CLK:=EN, Q=>);

IF pulse.Q THEN
	//Si une autre fonction est déjà en cours de traitement (token déjà pris) le canal ne peut pas être ouvert
	//La variable run garde l'ordre d'activation en mémoire et ouvre le canal dès que le token est libéré
	run := TRUE;
END_IF

IF run THEN 
	IF _start_communication(started := started) THEN 	// Vérifie si le token est libre
		G_DXL.usiFonction := G_DXL.usiGET_PRESENT_LOAD;	// configure le canal à ouvrir
		G_DXL.bRun := TRUE;								// envoie la commande au script python
		load := G_DXL.iDxl_load;						// si le canal est ouvert, renvoie la valeur actuelle du torque émit pas le moteur
	END_IF
	IF NOT EN THEN
		G_DXL.bRun 	:= FALSE;						    //ferme le canal
		G_DXL.iDxl_load := -9000;						//remet une valeur par défault
		_end_communication(run:=run,started := started);//libère le token
	END_IF;
ELSE
	load := -9000;										//valeur par défaut
END_IF
END_METHOD

METHOD get_movement 
VAR_INPUT
	EN:BOOL; 	// ouvre un canal de transmission avec le moteur 
END_VAR
VAR_OUTPUT
	mouvement:BOOL; // le moteur renvoie si il est en mouvement(TRUE) ou non (FALSE)
END_VAR
VAR_INST 
	run :BOOL;
	pulse : R_TRIG;
	started: BOOL;
END_VAR
//ouvre le canal de transmission
pulse(CLK:=EN, Q=>);

IF pulse.Q THEN
	//Si une autre fonction est déjà en cours de traitement (token déjà pris) le canal ne peut pas être ouvert
	//La variable run garde l'ordre d'activation en mémoire et ouvre le canal dès que le token est libéré
	run := TRUE;
END_IF

IF run THEN 
	IF _start_communication(started := started) THEN 	// Vérifie si le token est libre
		G_DXL.usiFonction := G_DXL.usiGET_PRESENT_MOVEMENT;	// configure le canal à ouvrir
		G_DXL.bRun := TRUE;								// envoie la commande au script python
		mouvement := G_DXL.bDxl_movement;				// status du mouvement du moteur Dynamixel
	END_IF
	IF NOT EN THEN
		G_DXL.bRun 	:= FALSE;						    //ferme le canal
		G_DXL.bDxl_movement := 1;						//remet une valeur par défault
		_end_communication(run:=run,started := started);//libère le token
	END_IF;
ELSE
	mouvement := 1;										//valeur par défaut
END_IF
END_METHOD

METHOD get_position
VAR_INPUT
	EN:BOOL; 	// ouvre un canal de transmission avec le moteur 
END_VAR
VAR_OUTPUT
	position:DINT; //(AX12A sur 300 degrés)0-1023 ou (XL430 sur 360 degrés)0-4095 ou (XL430 en multitours)+- 1'048'575
END_VAR
VAR_INST 
	run :BOOL;
	pulse : R_TRIG;
	started: BOOL;
END_VAR
//ouvre le canal de transmission
pulse(CLK:=EN, Q=>);

IF pulse.Q THEN
	//Si une autre fonction est déjà en cours de traitement (token déjà pris) le canal ne peut pas être ouvert
	//La variable run garde l'ordre d'activation en mémoire et ouvre le canal dès que le token est libéré
	run := TRUE;
END_IF

IF run THEN 
	IF _start_communication(started := started) THEN 	// Vérifie si le token est libre
		G_DXL.usiFonction := G_DXL.usiGET_PRESENT_POSITION;	// configure le canal à ouvrir
		G_DXL.bRun := TRUE;								// envoie la commande au script python
		position := G_DXL.diDxl_position;				//(AX12A sur 300 degrés)0-1023 ou (XL430 sur 360 degrés)0-4095 ou (XL430 en multitours)+- 1'048'575
	END_IF
	IF NOT EN THEN
		G_DXL.bRun 	:= FALSE;						    //ferme le canal
		G_DXL.diDxl_position := -9000;					//remet une valeur par défault
		_end_communication(run:=run,started := started);//libère le token
	END_IF;
ELSE
	position := -9000;									//valeur par défaut
END_IF
END_METHOD

METHOD send_acceleration 
VAR_INPUT
	EN			:BOOL; // un front montant change le taux d'accélération du moteur
	acceleration:USINT;// acceleration de 0-100 (100 => acceleration instantanée)
	speed		:INT:=32767; // vitesse de pointe 0-32767
END_VAR
VAR_OUTPUT
	done		:BOOL; //la commande est envoyée, passe à False si EN passe aussi à False
END_VAR
VAR_INST 
	bRun 		:BOOL;
	rtrigPulse 	:R_TRIG;
	bDone_pulse :BOOL;
	bStarted 	:BOOL;
END_VAR
//Activation de la fonction
rtrigPulse(CLK:=EN, Q=>);

IF rtrigPulse.Q THEN
	//Si une autre fonction est déjà en cours de traitement (token déjà pris) cette fonction ne peut pas être effectuée
	//La variable run garde l'ordre d'activation en mémoire et lance la fonction dès que le token est libéré
	bRun := TRUE;
END_IF

IF bRun THEN
	IF _start_communication(started:=bStarted) THEN 								//vérifie si les tokens sont libérés 
		G_DXL.usiFonction := G_DXL.usiGOAL_ACCELERATION;								//Ecriture de la commande
		G_DXL.usiAcceleration := acceleration;
		G_DXL.iSpeed    := speed;
		bDone_pulse := _end_communication(run:=bRun, started:=bStarted) AND EN;	//libère le token une fois que la commande est lancée
		_send();																//Envoi de la commande au moteur
	END_IF
END_IF;

IF bDone_pulse AND EN THEN														//Affiche le status d'excution de la fonction
	done := EN;																	//tant que EN est à True
ELSIF bDone_pulse AND NOT EN THEN
	bDone_pulse := FALSE;
END_IF
END_METHOD

METHOD send_disable_torque
VAR_INPUT
	EN			:BOOL; // un front montant désactive le torque du moteur 
END_VAR
VAR_OUTPUT
	done		:BOOL; //la commande est envoyée, passe à False si EN passe aussi à False
END_VAR
VAR_INST 
	run 		:BOOL;
	pulse 		:R_TRIG;
	done_pulse 	:BOOL;
	started 	:BOOL;
END_VAR
//Activation de la fonction
pulse(CLK:=EN, Q=>);

IF pulse.Q THEN
	//Si une autre fonction est déjà en cours de traitement (token déjà pris) cette fonction ne peut pas être effectuée
	//La variable run garde l'ordre d'activation en mémoire et lance la fonction dès que le token est libéré
	run := TRUE;
END_IF

IF run THEN
	IF _start_communication(started:=started) THEN 								//vérifie si les tokens sont libérés 
		G_DXL.usiFonction := G_DXL.usiDISABLE_TORQUE;									//Ecriture de la commande
		done_pulse := _end_communication(run:=run, started:=started) AND EN;	//libère le token une fois que la commande est lancée
		_send();																//Envoi de la commande au moteur
	END_IF
END_IF;

IF done_pulse AND EN THEN														//Affiche le status d'excution de la fonction
	done := EN;																	//tant que EN est à True
ELSIF done_pulse AND NOT EN THEN
	done_pulse := FALSE;
END_IF
END_METHOD

METHOD send_enable_torque 
VAR_INPUT
	EN			:BOOL; // un front montant active le torque du moteur 
END_VAR
VAR_OUTPUT
	done		:BOOL; //la commande est envoyée, passe à False si EN passe aussi à False
END_VAR
VAR_INST 
	run 		:BOOL;
	pulse 		:R_TRIG;
	done_pulse 	:BOOL;
	started 	:BOOL;
END_VAR
//Activation de la fonction
pulse(CLK:=EN, Q=>);

IF pulse.Q THEN
	//Si une autre fonction est déjà en cours de traitement (token déjà pris) cette fonction ne peut pas être effectuée
	//La variable run garde l'ordre d'activation en mémoire et lance la fonction dès que le token est libéré
	run := TRUE;
END_IF

IF run THEN
	IF _start_communication(started:=started) THEN 								//vérifie si les tokens sont libérés 
		G_DXL.usiFonction := G_DXL.usiENABLE_TORQUE;									//Ecriture de la commande
		done_pulse := _end_communication(run:=run, started:=started) AND EN;	//libère le token une fois que la commande est lancée
		_send();																//Envoi de la commande au moteur
	END_IF
END_IF;

IF done_pulse AND EN THEN														//Affiche le status d'excution de la fonction
	done := EN;																	//tant que EN est à True
ELSIF done_pulse AND NOT EN THEN
	done_pulse := FALSE;
END_IF
END_METHOD

METHOD send_led_off 
VAR_INPUT
	EN			:BOOL; // un front montant éteint la led
END_VAR
VAR_OUTPUT
	done		:BOOL; //la commande est envoyée, passe à False si EN passe aussi à False
END_VAR
VAR_INST 
	run 		:BOOL;
	pulse 		:R_TRIG;
	done_pulse 	:BOOL;
	started 	:BOOL;
END_VAR
//Activation de la fonction
pulse(CLK:=EN, Q=>);

IF pulse.Q THEN
	//Si une autre fonction est déjà en cours de traitement (token déjà pris) cette fonction ne peut pas être effectuée
	//La variable run garde l'ordre d'activation en mémoire et lance la fonction dès que le token est libéré
	run := TRUE;
END_IF

IF run THEN
	IF _start_communication(started:=started) THEN 								//vérifie si les tokens sont libérés 
		G_DXL.usiFonction := G_DXL.usiLED_OFF;										//Ecriture de la commande
		done_pulse := _end_communication(run:=run, started:=started) AND EN;	//libère le token une fois que la commande est lancée
		_send();																//Envoi de la commande au moteur
	END_IF
END_IF;

IF done_pulse AND EN THEN														//Affiche le status d'excution de la fonction
	done := EN;																	//tant que EN est à True
ELSIF done_pulse AND NOT EN THEN
	done_pulse := FALSE;
END_IF
END_METHOD

METHOD send_led_on 
VAR_INPUT
	EN			:BOOL; // un front montant allume la led
END_VAR
VAR_OUTPUT
	done		:BOOL; //la commande est envoyée, passe à False si EN passe aussi à False
END_VAR
VAR_INST 
	run 		:BOOL;
	pulse 		:R_TRIG;
	done_pulse 	:BOOL;
	started 	:BOOL;
END_VAR
//Activation de la fonction
pulse(CLK:=EN, Q=>);

IF pulse.Q THEN
	//Si une autre fonction est déjà en cours de traitement (token déjà pris) cette fonction ne peut pas être effectuée
	//La variable run garde l'ordre d'activation en mémoire et lance la fonction dès que le token est libéré
	run := TRUE;
END_IF

IF run THEN
	IF _start_communication(started:=started) THEN 								//vérifie si les tokens sont libérés 
		G_DXL.usiFonction := G_DXL.usiLED_ON;											//Ecriture de la commande
		done_pulse := _end_communication(run:=run, started:=started) AND EN;	//libère le token une fois que la commande est lancée
		_send();																//Envoi de la commande au moteur
	END_IF
END_IF;

IF done_pulse AND EN THEN														//Affiche le status d'excution de la fonction
	done := EN;																	//tant que EN est à True
ELSIF done_pulse AND NOT EN THEN
	done_pulse := FALSE;
END_IF
END_METHOD

METHOD send_operating_mode 
VAR_INPUT
	EN			:BOOL; // active la fonction
	mode		:STRING; //‘position’ ou ‘position_angleMin_angleMax’ ou ‘extended position’ ou‘velocity' ou ‘PWM’ 
END_VAR
VAR_OUTPUT
	done		:BOOL; //la commande est envoyée, passe à False si EN passe aussi à False
END_VAR
VAR_INST 
	run 		:BOOL;
	pulse 		:R_TRIG;
	done_pulse 	:BOOL;
	started 	:BOOL;
END_VAR
//Activation de la fonction
pulse(CLK:=EN, Q=>);

IF pulse.Q THEN
	//Si une autre fonction est déjà en cours de traitement (token déjà pris) cette fonction ne peut pas être effectuée
	//La variable run garde l'ordre d'activation en mémoire et lance la fonction dès que le token est libéré
	run := TRUE;
END_IF

IF run THEN
	IF _start_communication(started:=started) THEN 								//vérifie si les tokens sont libérés 
		G_DXL.usiFonction := G_DXL.usiOPERATING_MODE;									//Ecriture de la commande
		G_DXL.sMode := mode;
		done_pulse := _end_communication(run:=run, started:=started) AND EN;	//libère le token une fois que la commande est lancée
		_send();																//Envoi de la commande au moteur
	END_IF
END_IF;

IF done_pulse AND EN THEN														//Affiche le status d'excution de la fonction
	done := EN;																	//tant que EN est à True
ELSIF done_pulse AND NOT EN THEN
	done_pulse := FALSE;
END_IF
END_METHOD

METHOD send_position 
VAR_INPUT
	EN			:BOOL; // un front montant donne une nouvelle position au moteur à atteindre 
	position	:DINT; //(AX12A sur 300 degrés)0-1023 ou (XL430 sur 360 degrés)0-4095 ou (XL430 en multitours)+- 1'048'575
	vitesse		:INT;  //(AX12A)0-1023 ou (XL430)0-1023 
END_VAR
VAR_OUTPUT
	done		:BOOL; //la commande est envoyée, passe à False si EN passe aussi à False
END_VAR
VAR_INST 
	run 		:BOOL;
	pulse 		:R_TRIG;
	done_pulse 	:BOOL;
	started 	:BOOL;
END_VAR
//Activation de la fonction
pulse(CLK:=EN, Q=>);

IF pulse.Q THEN
	//Si une autre fonction est déjà en cours de traitement (token déjà pris) cette fonction ne peut pas être effectuée
	//La variable run garde l'ordre d'activation en mémoire et lance la fonction dès que le token est libéré
	run := TRUE;
END_IF

IF run THEN
	IF _start_communication(started:=started) THEN 								//vérifie si les tokens sont libérés 
		G_DXL.usiFonction := G_DXL.usiGOAL_POSITION;									//Ecriture de la commande
		G_DXL.diPosition := position;
		G_DXL.iSpeed    := vitesse;
		done_pulse := _end_communication(run:=run, started:=started) AND EN;	//libère le token une fois que la commande est lancée
		_send();																//Envoi de la commande au moteur
	END_IF
END_IF;

IF done_pulse AND EN THEN														//Affiche le status d'excution de la fonction
	done := EN;																	//tant que EN est à True
ELSIF done_pulse AND NOT EN THEN
	done_pulse := FALSE;
END_IF
END_METHOD

METHOD send_reset_position 
VAR_INPUT
	EN			:BOOL; // un front montant réinitialise la position du moteur sur 360 degrés
END_VAR
VAR_OUTPUT
	done		:BOOL; //la commande est envoyée, passe à False si EN passe aussi à False
END_VAR
VAR_INST 
	run 		:BOOL;
	pulse 		:R_TRIG;
	done_pulse 	:BOOL;
	started 	:BOOL;
END_VAR
//Activation de la fonction
pulse(CLK:=EN, Q=>);

IF pulse.Q THEN
	//Si une autre fonction est déjà en cours de traitement (token déjà pris) cette fonction ne peut pas être effectuée
	//La variable run garde l'ordre d'activation en mémoire et lance la fonction dès que le token est libéré
	run := TRUE;
END_IF

IF run THEN
	IF _start_communication(started:=started) THEN 								//vérifie si les tokens sont libérés 
		G_DXL.usiFonction := G_DXL.usiRESET_POSITION;									//Ecriture de la commande
		done_pulse := _end_communication(run:=run, started:=started) AND EN;	//libère le token une fois que la commande est lancée
		_send();																//Envoi de la commande au moteur
	END_IF
END_IF;

IF done_pulse AND EN THEN														//Affiche le status d'excution de la fonction
	done := EN;																	//tant que EN est à True
ELSIF done_pulse AND NOT EN THEN
	done_pulse := FALSE;
END_IF
END_METHOD

METHOD send_stop_position 
VAR_INPUT
	EN			:BOOL; // un front montant arrête le moteur à sa position actuelle
	reset 		:BOOL; // reset la position 
END_VAR
VAR_OUTPUT
	done		:BOOL; //la commande est envoyée, passe à False si EN passe aussi à False
END_VAR
VAR_INST 
	run 		:BOOL;
	pulse 		:R_TRIG;
	done_pulse 	:BOOL;
	started 	:BOOL;
END_VAR
//Activation de la fonction
pulse(CLK:=EN, Q=>);

IF pulse.Q THEN
	//Si une autre fonction est déjà en cours de traitement (token déjà pris) cette fonction ne peut pas être effectuée
	//La variable run garde l'ordre d'activation en mémoire et lance la fonction dès que le token est libéré
	run := TRUE;
END_IF

IF run THEN
		IF _start_communication(started:=started) THEN 								//vérifie si les tokens sont libérés 
		G_DXL.usiFonction := G_DXL.usiSTOP_POSITION;										//Ecriture de la commande
		G_DXL.bReset	   := reset;
		done_pulse := _end_communication(run:=run, started:=started) AND EN;		//libère le token une fois que la commande est lancée
		_send();																	//Envoi de la commande au moteur
	END_IF
END_IF;

IF done_pulse AND EN THEN														//Affiche le status d'excution de la fonction
	done := EN;																	//tant que EN est à True
ELSIF done_pulse AND NOT EN THEN
	done_pulse := FALSE;
END_IF
END_METHOD

METHOD send_velocity 
VAR_INPUT
	EN			:BOOL; // un front montant donne une nouvelle vitesse au moteur en mode velocity
	vitesse		:INT;  //(XL430)+-1023 
END_VAR
VAR_OUTPUT
	done		:BOOL; //la commande est envoyée, passe à False si EN passe aussi à False
END_VAR
VAR_INST 
	run 		:BOOL;
	pulse 		:R_TRIG;
	done_pulse 	:BOOL;
	started 	:BOOL;
END_VAR
//Activation de la fonction
pulse(CLK:=EN, Q=>);

IF pulse.Q THEN
	//Si une autre fonction est déjà en cours de traitement (token déjà pris) cette fonction ne peut pas être effectuée
	//La variable run garde l'ordre d'activation en mémoire et lance la fonction dès que le token est libéré
	run := TRUE;
END_IF

IF run THEN
	IF _start_communication(started:=started) THEN 								//vérifie si les tokens sont libérés 
		G_DXL.usiFonction := G_DXL.usiGOAL_VELOCITY;									//Ecriture de la commande
		G_DXL.iSpeed    := vitesse;
		done_pulse := _end_communication(run:=run, started:=started) AND EN;	//libère le token une fois que la commande est lancée
		_send();																//Envoi de la commande au moteur
	END_IF
END_IF;

IF done_pulse AND EN THEN														//Affiche le status d'excution de la fonction
	done := EN;																	//tant que EN est à True
ELSIF done_pulse AND NOT EN THEN
	done_pulse := FALSE;
END_IF
END_METHOD

END_FUNCTION_BLOCK

// ---- POUs/Utillity/Maths/RAD2DEGRE.TcPOU
FUNCTION RAD2DEGRE : lreal
VAR_INPUT
	lrAngle : LREAL;
END_VAR
VAR
END_VAR

RAD2DEGRE := lrAngle*180/PI;

END_FUNCTION

// ---- POUs/Utillity/Structure/Tableau/AddStep.TcPOU
FUNCTION AddStep : bool
VAR_INPUT
	step:ST_Tableau;
END_VAR
VAR
	icounter:INT;
	etapeSuivante:INT;
END_VAR

//ajoute une étape après
etapeSuivante := G_Match.iLigne+1;
FOR icounter := 100 TO etapeSuivante BY -1 DO
  G_Match.Tableau[icounter] := G_Match.Tableau[icounter-1];
END_FOR 
G_Match.Tableau[etapeSuivante] := step;

END_FUNCTION

// ---- POUs/Utillity/Structure/Tableau/PointsRestants.TcPOU
FUNCTION PointsRestants : INT
VAR_INPUT
END_VAR
VAR
	icounter:INT;
	points:INT;
END_VAR

//calcul le nombre de points restant jusqu'à la prochaine étape nommée
FOR icounter := G_Match.iLigne TO 100 BY 1 DO
	points := points + G_Match.Tableau[G_Match.iCounter].uiAjoutPoints_pts;
	IF G_Match.Tableau[G_Match.iCounter].NomEtape <> '' THEN
		EXIT;
	END_IF
END_FOR
PointsRestants := points;

END_FUNCTION

// ---- GlobalTextList.TcGTLO
TEXTLIST GlobalTextList
  386 = ' Init Position'
  863 = '%'
  858 = '%10.0f'
  354 = '%10.1f'
  311 = '%s'
  35 = '%t[m.ss]'
  38 = '0°'
  36 = '180°'
  37 = '270°'
  33 = '90°'
  302 = 'Accel.'
  105 = 'Accél.'
  939 = 'Accélération'
  782 = 'Action tes'
  547 = 'Action test'
  859 = 'Actionneur'
  823 = 'Activation balise'
  1171 = 'activer mode test'
  142 = 'Angle'
  42 = 'Angle 1 : Nothing'
  30 = 'Angle 2 : %10.1f'
  40 = 'Angle 2 : Nothing'
  1261 = 'Angle 3 : %10.1f'
  1278 = 'Angle 3 : Nothing'
  12 = "Angle d'approche"
  29 = 'Angle1 : %10.1f'
  34 = 'Arrêt détection'
  330 = 'Atelier | Bureau'
  629 = 'Balise'
  591 = 'Barillet'
  43 = 'bloquage roue'
  728 = 'Bloquage Roue'
  761 = 'Burean  | Atelierprogression'
  555 = 'Bureau | Atelier'
  451 = 'Bureau | Python'
  659 = 'Chronomètre:'
  948 = 'Config'
  145 = 'Config Mode'
  2 = 'Config Moe'
  45 = 'Deccel.'
  401 = 'Deplacement'
  41 = 'Distance 1 : Nothing'
  39 = 'Distance 2 : Nothing'
  1269 = 'Distance 3 : Nothing'
  28 = 'Distance1 : %10.1f'
  32 = 'Distance2 : %10.1f'
  1252 = 'Distance3 : %10.1f'
  368 = 'Décél.'
  1054 = 'Décélération'
  827 = 'erreur'
  653 = 'Fin Match'
  1287 = 'GENTIL'
  102 = 'G_Visus.sTestFunction2'
  1004 = 'Homologation'
  402 = 'INIT'
  432 = 'Init'
  778 = 'Init Barillet'
  572 = 'Init Bras'
  660 = 'Init Position'
  458 = 'Init progression'
  261 = 'Kimagure'
  174 = 'Led Bleu'
  732 = 'Led Rouge'
  749 = 'Led Vert'
  573 = 'Machibuse'
  408 = 'marche arrière'
  463 = 'Marche arrière'
  932 = 'Match '
  1113 = 'Match en cours'
  171 = 'Menu'
  0 = 'Moteur power'
  1244 = 'Méchant'
  44 = 'Méchant 1'
  160 = 'Méchant 2'
  86 = 'Méchant 3'
  657 = 'Oikake'
  731 = 'Otoboke'
  448 = 'Panneau Commande'
  617 = 'Parcours 1'
  580 = 'Parcours 2'
  619 = 'Parcours 3'
  182 = 'Points'
  68 = 'Points :'
  1030 = 'Points :;'
  968 = 'Pompe'
  76 = 'position'
  544 = 'Position X'
  675 = 'Position Y'
  180 = 'Position Z'
  139 = 'Prematch'
  651 = 'prêt pour start'
  81 = 'python'
  424 = 'Radio Button'
  464 = 'Reset'
  47 = 'reset pos'
  691 = 'Reset position'
  58 = 'Restart'
  665 = 'RETOUR'
  567 = 'Retour'
  132 = 'robot en 0'
  678 = 'roue bloqué'
  87 = 'Run'
  595 = 'réelle'
  31 = 'start'
  214 = 'Start'
  658 = 'Start\nmatch'
  228 = 'Start Init'
  813 = 'Start Prematch'
  789 = 'Start python'
  773 = 'Stop python'
  176 = 'Teams'
  638 = 'Test'
  848 = 'Visu_Balise'
  266 = 'Visu_Deplacement'
  365 = 'Visu_Test'
  924 = 'Vitesse'
  1073 = 'X'
  1018 = 'Y'
END_TEXTLIST

// ---- VISUs/Visu pour debug/V_Balise.TcVIS
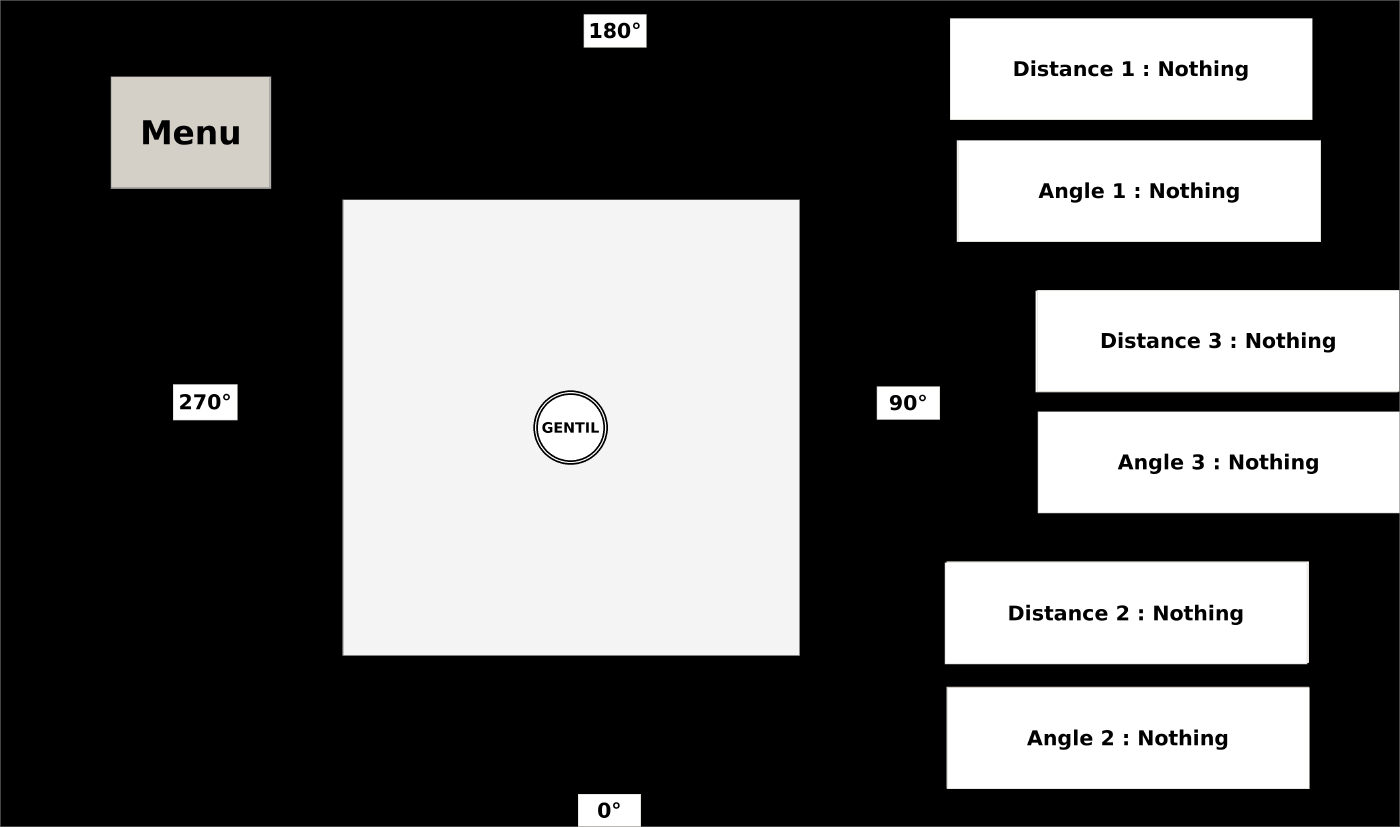
VISUALIZATION V_Balise  // 2454x1451
    Line (1000,750) (1000,50)
    Line (1000,750) (1700,750)
    Line (1000,750) (300,750)
    Line (1000,750) (1000,1450)
    Textfield (1665,32 635x178), "Distance1 : %10.1f", text variable: G_Balise.lrDistance_1, invisible if: ITInterruption.balise.Nothing1
    Textfield (1677,246 635x178), "Angle1 : %10.1f", text variable: G_Balise.lrAngle_1, invisible if: ITInterruption.balise.Nothing1
    Textfield (1659,1205 635x178), "Angle 2 : %10.1f", text variable: G_Balise.lrAngle_2, invisible if: ITInterruption.balise.Nothing2
    Textfield (1659,985 635x178), "Distance2 : %10.1f", text variable: G_Balise.lrDistance_2, invisible if: ITInterruption.balise.Nothing2
    Textfield (1537,678 110x58), "90°", colour toggle: ITInterruption.balise.Angle90deg
    Textfield (1023,25 110x58), "180°", colour toggle: ITInterruption.balise.Angle180deg
    Textfield (303,674 113x63), "270°", colour toggle: ITInterruption.balise.Angle270deg
    Textfield (1013,1393 110x58), "0°", colour toggle: ITInterruption.balise.Angle0deg
    Textfield (1656,987 635x178), "Distance 2 : Nothing", text variable: G_Balise.lrDistance_2, invisible if: not ITInterruption.balise.Nothing2
    Textfield (1665,32 635x178), "Distance 1 : Nothing", text variable: G_Balise.lrDistance_1, invisible if: not ITInterruption.balise.Nothing1
    Pie (600,350 800x800), invisible if: ITInterruption.balise.Angle0deg
    Pie (600,350 800x800), invisible if: ITInterruption.balise.Angle90deg
    Pie (602,350 800x800), invisible if: ITInterruption.balise.Angle180deg
    Pie (601,350 800x800), invisible if: ITInterruption.balise.Angle270deg
    Ellipse (935,685 130x130), "Méchant", invisible if: ITInterruption.balise.Nothing2
        p3528305787: ITInterruption.balise.posiX2
        p2773130477: ITInterruption.balise.posiY2
        p874137650: ITInterruption.balise.posiX2
        p1126004900: ITInterruption.balise.posiY2
    Ellipse (935,685 130x130), "Méchant", invisible if: ITInterruption.balise.Nothing1
        p3528305787: ITInterruption.balise.posiX1
        p2773130477: ITInterruption.balise.posiY1
        p874137650: ITInterruption.balise.posiX1
        p1126004900: ITInterruption.balise.posiY1
    Line (1000,750) (1000,750), colour toggle: ITInterruption.balise.D1_40cm, invisible if: ITInterruption.balise.Nothing1
        p874137650: ITInterruption.balise.posiX1
        p1126004900: ITInterruption.balise.posiY1
    Line (1000,750) (1000,750), colour toggle: ITInterruption.balise.D2_40cm, invisible if: ITInterruption.balise.Nothing2
        p874137650: ITInterruption.balise.posiX2
        p1126004900: ITInterruption.balise.posiY2
    Textfield (1815,510 635x178), "Distance3 : %10.1f", text variable: G_Balise.ArrayEnnemi [2,1], invisible if: ITInterruption.balise.Nothing3
    Textfield (1819,722 635x178), "Angle 3 : %10.1f", text variable: G_Balise.lrAngle_2, invisible if: ITInterruption.balise.Nothing3
    Textfield (1818,509 635x178), "Distance 3 : Nothing", text variable: G_Balise.lrDistance_3, invisible if: not ITInterruption.balise.Nothing3
    Ellipse (935,685 130x130), "Méchant", invisible if: ITInterruption.balise.Nothing3
        p3528305787: ITInterruption.balise.posiX3
        p2773130477: ITInterruption.balise.posiY3
        p874137650: ITInterruption.balise.posiX3
        p1126004900: ITInterruption.balise.posiY3
    Line (1000,750) (1000,750), colour toggle: ITInterruption.balise.D3_40cm, invisible if: ITInterruption.balise.Nothing3
        p874137650: ITInterruption.balise.posiX3
        p1126004900: ITInterruption.balise.posiY3
    Ellipse (940,690 120x120), "GENTIL"
    Textfield (1819,722 635x178), "Angle 3 : Nothing", text variable: G_Balise.lrAngle_3, invisible if: not ITInterruption.balise.Nothing3
    Textfield (1680,246 635x178), "Angle 1 : Nothing", text variable: G_Balise.lrAngle_1, invisible if: not ITInterruption.balise.Nothing1
    Textfield (1660,1206 635x178), "Angle 2 : Nothing", text variable: G_Balise.lrAngle_2, invisible if: not ITInterruption.balise.Nothing2
    Button (194,134 281x197), "Menu"
        OnMouseDown: change screen: V_Menu
END_VISUALIZATION

// ---- VISUs/Visu pour debug/V_Config.TcVIS
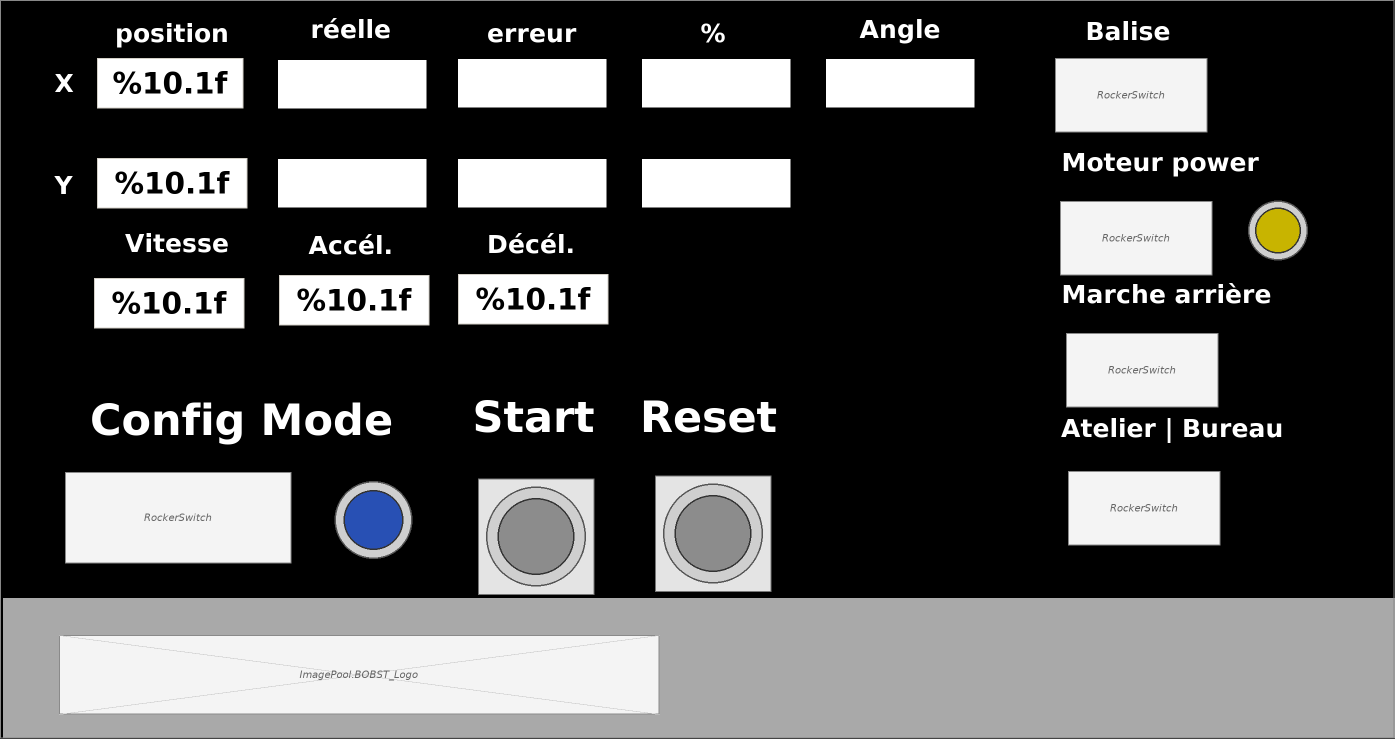
VISUALIZATION V_Config  // 1395x739
    Rectangle (3,598 1396x140)
    Rectangle (457,158 150x50), "%10.1f", text variable: G_Visus.lrConfigErreurY
    Label (97,8 150x50), "position"
    Label (276,4 150x50), "réelle"
    Label (457,8 150x50), "erreur"
    Label (663,8 100x50), "%"
    Textfield (97,58 146x50), "%10.1f", text variable: G_Visus.lrConfigPosX
        OnMouseDown: write G_Visus.lrConfigPosX via InputWithLimits, min 0, max 1000000
    Textfield (97,158 150x50), "%10.1f", text variable: G_Visus.lrConfigPosY
        OnMouseDown: write G_Visus.lrConfigPosY via InputWithLimits, min 0, max 3000
    Rectangle (277,59 150x50), "%10.1f", text variable: G_Odometrie.lrPositionX
    Rectangle (277,158 150x50), "%10.1f", text variable: G_Odometrie.lrPositionY
    Rectangle (457,58 150x50), "%10.1f", text variable: G_Visus.lrConfigErreurX
    Rectangle (641,58 150x50), "%10.1f", text variable: G_Visus.lrConfigErreurX_Pourcent
    Rectangle (641,158 150x50), "%10.1f", text variable: G_Visus.lrConfigErreurY_pourcent
    Label (40,58 49x50), "X"
    Label (39,160 49x50), "Y"
    Rectangle (825,58 150x50), "%10.1f", text variable: G_Odometrie.lrAngleDeg
    Label (825,4 150x50), "Angle"
    Textfield (94,278 150x50), "%10.1f", text variable: G_Visus.lrConfigVitesse
        OnMouseDown: write G_Visus.lrConfigVitesse via InputWithLimits, min 0, max 1700
    Label (102,218 150x50), "Vitesse"
    Label (258,220 186x50), "Accél."
    Label (429,219 204x50), "Décél."
    Textfield (279,275 150x50), "%10.1f", text variable: G_Visus.lrConfigAcc
        OnMouseDown: write G_Visus.lrConfigAcc via Default, min 0, max 1500
    Textfield (458,274 150x50), "%10.1f", text variable: G_Visus.lrConfigDecc
        OnMouseDown: write G_Visus.lrConfigDecc via InputWithLimits, min 0, max 1500
    RockerSwitch (1055,58 152x74), variable: G_Visus.bConfigBalise, behaviour: TOGGLE, style: Switch-RockerSwitch-Gray
    Label (1053,6 150x50), "Balise"
    RockerSwitch (65,472 226x91), variable: G_Visus.bConfigEnable, behaviour: TOGGLE, style: Switch-RockerSwitch-Gray
    Label (72,392 339x56), "Config Mode"
    Lamp1 (322,475 103x90), variable: G_Visus.bConfigReady, style: Lamp-Lamp1-Blue
    RockerSwitch (1060,201 152x74), variable: G_Visus.bConfigMoteurPower, behaviour: TOGGLE, style: Switch-RockerSwitch-Gray
    Label (1059,137 203x50), "Moteur power"
    Lamp1 (1242,196 72x69), variable: G_Visus.bConfigMoteurReady, style: Lamp-Lamp1-Yellow
    RockerSwitch (1066,333 152x74), variable: G_Visus.bConfigMarcheArriere, behaviour: TOGGLE, style: Switch-RockerSwitch-Gray
    Label (1065,269 203x50), "Marche arrière"
    PushSwitch (478,466 116x141), variable: G_Visus.bConfigStart, behaviour: TOGGLE, style: Switch-PushSwitch-Gray
    Label (447,392 173x50), "Start"
    PushSwitch (655,463 116x141), variable: G_Visus.bConfigReset, behaviour: TAP, style: Switch-PushSwitch-Gray
    Label (625,392 167x50), "Reset"
    Label (1064,403 217x50), "Atelier | Bureau"
    RockerSwitch (1068,471 152x74), variable: G_Visus.bConfigChoixCote, behaviour: TOGGLE, style: Switch-RockerSwitch-Gray
    Image (59,635 600x79), image: ImagePool.BOBST_Logo
        OnMouseDown: change screen: V_Menu
END_VISUALIZATION

// ---- VISUs/Visu pour debug/V_Deplacement.TcVIS
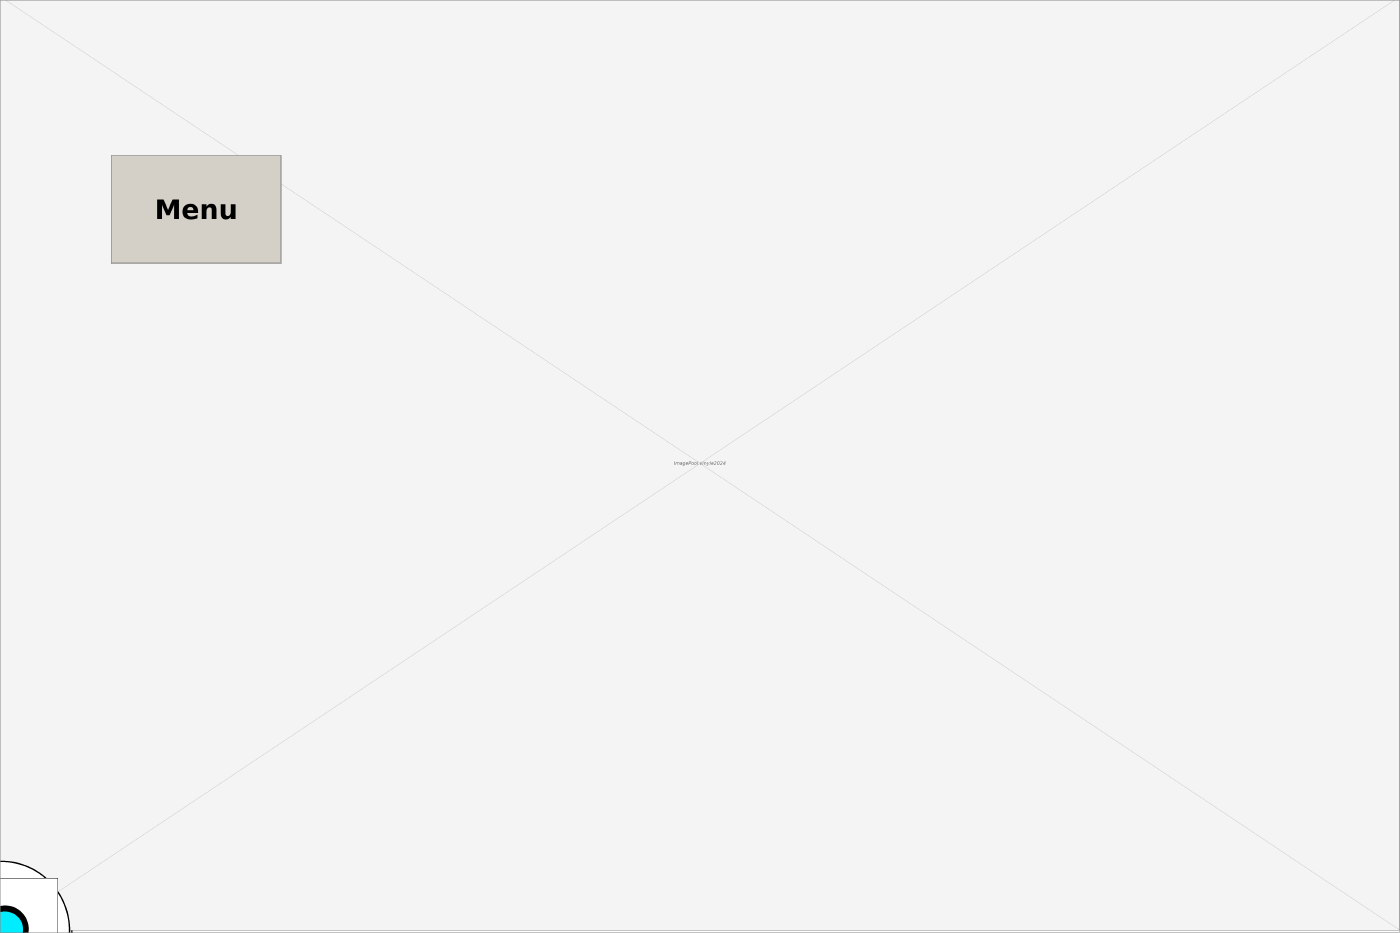
VISUALIZATION V_Deplacement  // 3000x2000
    Ellipse (-142,1844 294x300), "Méchant 1", invisible if: ITInterruption.balise.Nothing1
        p3560616238: ITInterruption.balise.CoordX1
        p2738717112: ITInterruption.balise.CoordY1
    Ellipse (-139,1841 294x300), "Méchant 3", invisible if: ITInterruption.balise.Nothing3
        p3560616238: ITInterruption.balise.CoordX3
        p2738717112: ITInterruption.balise.CoordY3
    Image (0,-8 3000x2002), image: ImagePool.vinyle2024
    Ellipse (-144,1845 294x300), "Méchant 2", invisible if: ITInterruption.balise.Nothing2
        p3560616238: ITInterruption.balise.CoordX2
        p2738717112: ITInterruption.balise.CoordY2
    RoundedRectangle (-102,1882 226x226)
        p2858320360: 360-G_Odometrie.lrAngleDeg
        p3560616238: G_Odometrie.lrPositionX
        p2738717112: -G_Odometrie.lrPositionY
    Ellipse (-39,1941 100x100)
        p3560616238: G_Odometrie.lrPositionX
        p2738717112: -G_Odometrie.lrPositionY
        p2858320360: 360-G_Odometrie.lrAngleDeg
    Ellipse (-74,2050 35x35)
        p3560616238: G_Odometrie.lrPositionX
        p2738717112: -G_Odometrie.lrPositionY
        p2858320360: 360-G_Odometrie.lrAngleDeg
    Button (238,333 365x232), "Menu"
        OnMouseDown: change screen: V_Menu
    Ellipse (-30,1953 80x78)
        p3560616238: ITMotion.odometrie.lrExpectedX
        p2738717112: -ITMotion.odometrie.lrExpectedY
END_VISUALIZATION

// ---- VISUs/Visu pour debug/V_Test.TcVIS
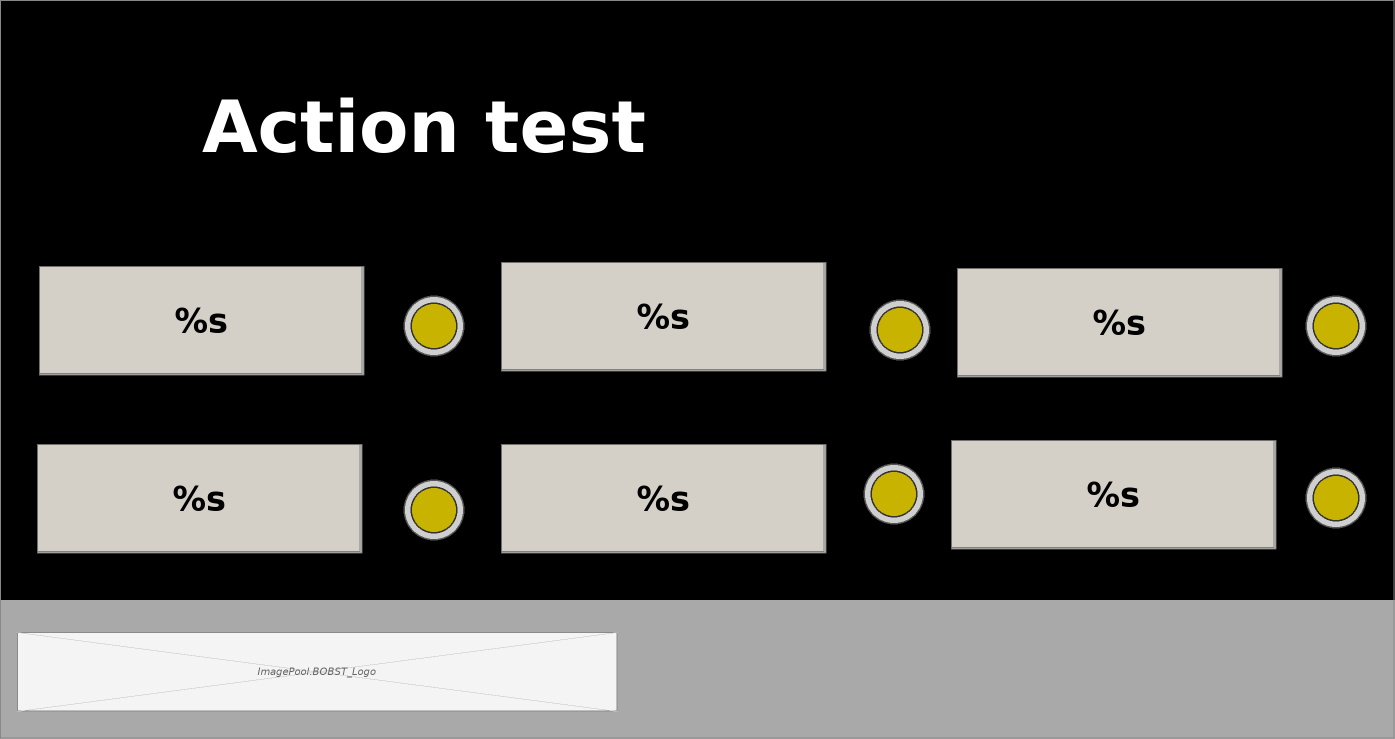
VISUALIZATION V_Test  // 1395x739
    Rectangle (-1,600 1396x140)
    Image (17,632 600x79), image: ImagePool.BOBST_Logo
        OnMouseDown: change screen: V_Menu
    Button (39,266 325x109), "%s", text variable: G_Visus.sTestFunction1
        OnMouseClick: execute { G_Visus.sTestBouton1 := True; }
    Button (501,262 325x109), "%s", text variable: G_Visus.sTestFunction2
        OnMouseClick: execute { G_Visus.sTestBouton2 := True; }
    Button (957,268 325x109), "%s", text variable: G_Visus.sTestFunction3
        OnMouseClick: execute { G_Visus.sTestBouton3 := True; }
    Button (37,444 325x109), "%s", text variable: G_Visus.sTestFunction4
        OnMouseClick: execute { G_Visus.sTestBouton4 := True; }
    Button (501,444 325x109), "%s", text variable: G_Visus.sTestFunction5
        OnMouseClick: execute { G_Visus.sTestBouton5 := True; }
    Button (951,440 325x109), "%s", text variable: G_Visus.sTestFunction6
        OnMouseClick: execute { G_Visus.sTestBouton6 := True; }
    Lamp1 (399,291 70x70), variable: G_Visus.sTestBouton1, style: Lamp-Lamp1-Yellow
    Lamp1 (865,295 70x70), variable: G_Visus.sTestBouton2, style: Lamp-Lamp1-Yellow
    Lamp1 (1301,291 70x70), variable: G_Visus.sTestBouton3, style: Lamp-Lamp1-Yellow
    Lamp1 (399,475 70x70), variable: G_Visus.sTestBouton4, style: Lamp-Lamp1-Yellow
    Lamp1 (859,459 70x70), variable: G_Visus.sTestBouton5, style: Lamp-Lamp1-Yellow
    Lamp1 (1301,463 70x70), variable: G_Visus.sTestBouton6, style: Lamp-Lamp1-Yellow
    Textfield (20,62 808x129), "Action test"
END_VISUALIZATION

// ---- VISUs/Visu pour match/V_Fin_Match.TcVIS
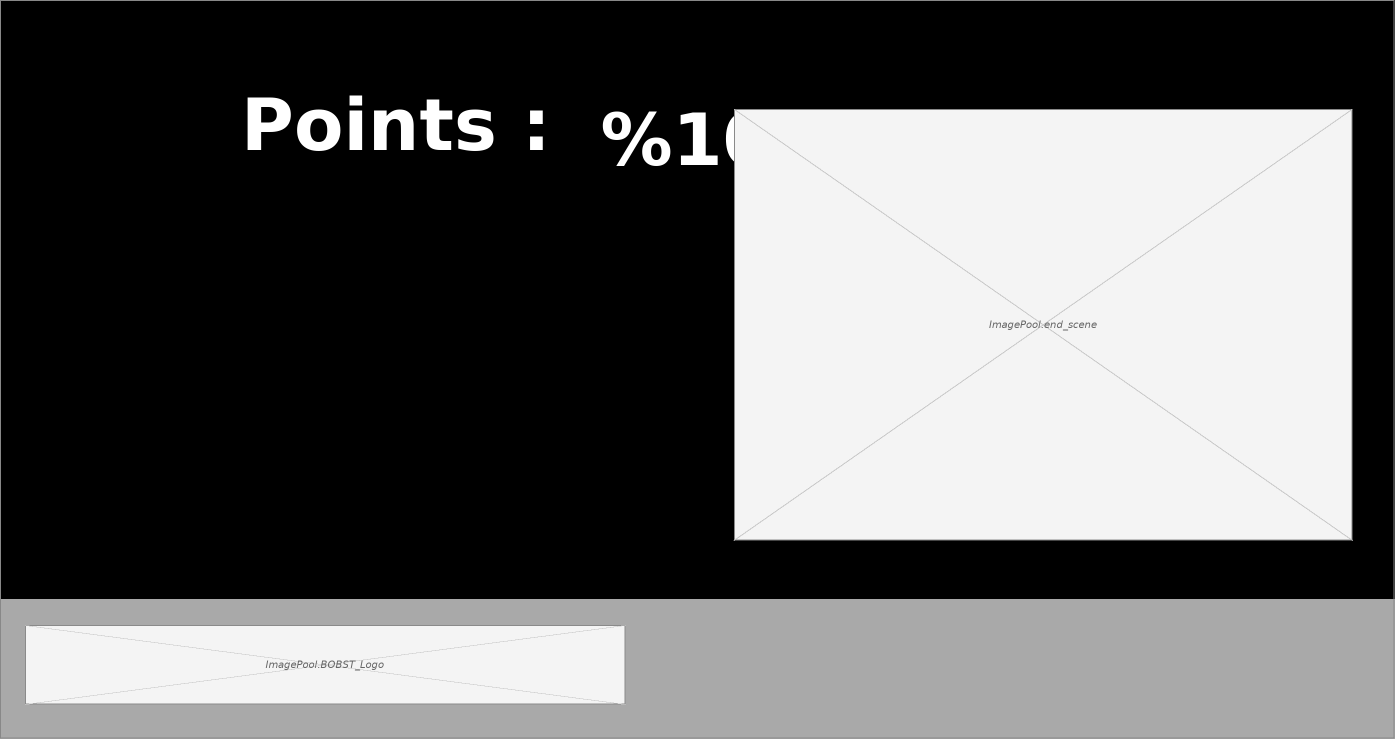
VISUALIZATION V_Fin_Match  // 1395x739
    Rectangle (0,599 1396x140)
    Textfield (516,75 450x129), "%10.0f", text variable: G_Match.PointMatch
    Textfield (158,60 476x129), "Points :"
    Image (25,625 600x79), image: ImagePool.BOBST_Logo
        OnMouseDown: change screen: V_Menu
    Image (734,109 618x431), image: ImagePool.end_scene
END_VISUALIZATION

// ---- VISUs/Visu pour match/V_Init.TcVIS
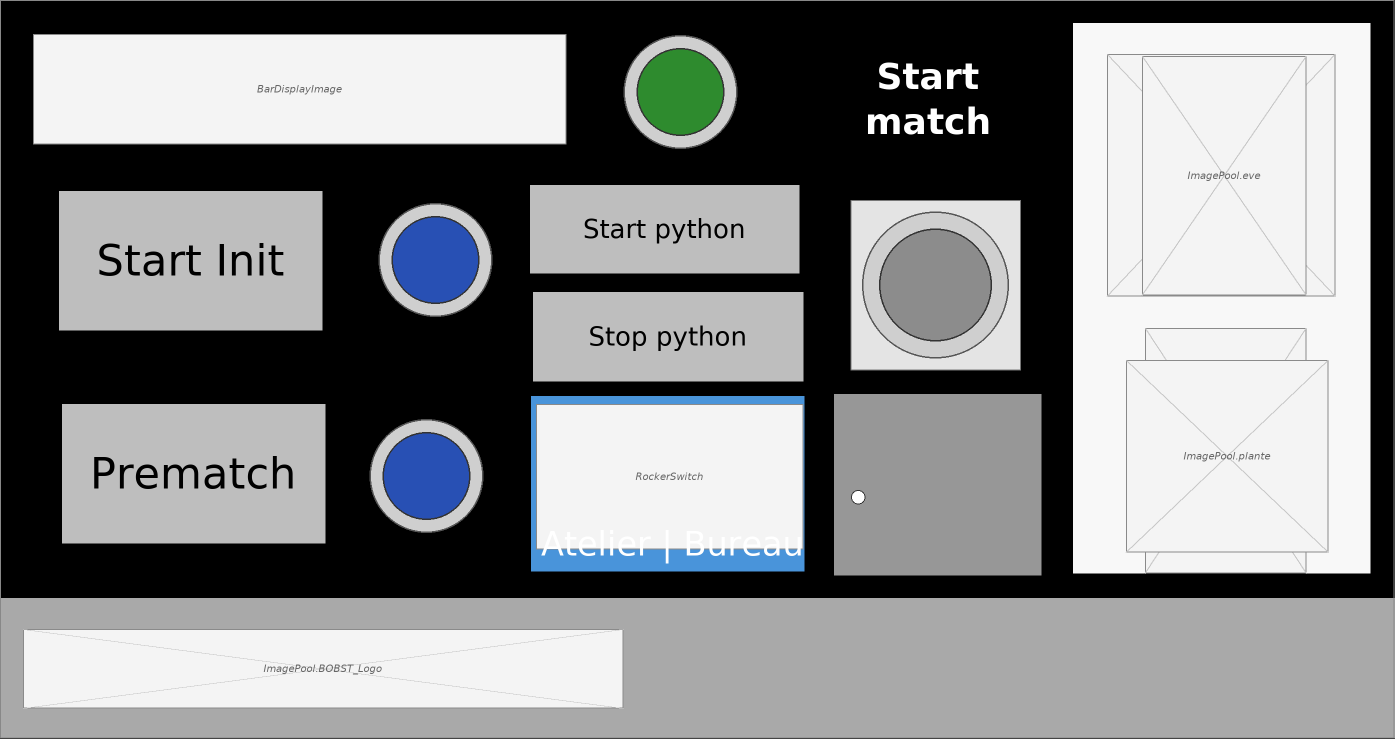
VISUALIZATION V_Init  // 1395x739
    Rectangle (-1,598 1396x140)
    RoundedRectangle (530,395 275x177)
    RoundedRectangle (1072,22 299x552)
    RoundedRectangle (833,393 209x183)
    Lamp1 (363,194 145x132), variable: G_init.ietapeInit <> 0, style: Lamp-Lamp1-Blue
    RockerSwitch (536,404 267x145), variable: G_Visus.bInitChoixCote, behaviour: TOGGLE, style: Switch-RockerSwitch-Gray
    BarDisplayImage (33,34 533x110), value: G_Visus.iInitProgressBar, style: BarDisplayImage-Gray, scale format: %.1f, scale 0..100
    Lamp1 (354,410 145x132), variable: G_PreMatch.bPrematchActive, style: Lamp-Lamp1-Blue
    Label (504,504 337x79), "Atelier | Bureau"
    RoundedRectangle (58,190 265x141), "Start Init"
        OnMouseDown: toggle G_Visus.bInitStart
        OnMouseUp: toggle G_Visus.bInitStart
    RoundedRectangle (61,403 265x141), "Prematch"
        OnMouseDown: toggle G_Visus.bInitPrematch
        OnMouseUp: toggle G_Visus.bInitPrematch
    RadioButton (849,432 178x130), variable: G_Visus.iInitChoixParcours
        Areas[0]: Text=Radiobutton
        Areas[1]: Text=Radiobutton
        p340057476: Parcours 1
        p3123465237: Parcours 2
        p2481256679: Parcours 3
    RoundedRectangle (1185,980 0x2)
    Lamp1 (608,26 145x132), variable: G_Visus.bInitPyScriptRunning, style: Lamp-Lamp1-Green
    RoundedRectangle (529,184 271x90), "Start python"
        OnMouseDown: toggle G_Visus.bInitStartPyscript
        OnMouseUp: toggle G_Visus.bInitStartPyscript
    RoundedRectangle (532,291 272x91), "Stop python"
        OnMouseDown: toggle G_Visus.bInitStopPyscript
        OnMouseUp: toggle G_Visus.bInitStopPyscript
    PushSwitch (849,200 173x170), variable: G_Visus.bInitStartMatch, behaviour: TAP, style: Switch-PushSwitch-Gray
    Label (835,47 186x104), "Start match"
    Image (23,629 600x79), image: ImagePool.BOBST_Logo
        OnMouseDown: change screen: V_Menu
    Image (1107,54 228x242), invisible if: G_Visus.bInitChoixCote, image: ImagePool.walle
    Image (1142,56 164x239), invisible if: not G_Visus.bInitChoixCote, image: ImagePool.eve
    Image (1145,328 161x245), invisible if: G_Visus.iInitChoixParcours = 1, image: ImagePool.botte
    Image (1126,360 202x192), invisible if: G_Visus.iInitChoixParcours = 0, image: ImagePool.plante
END_VISUALIZATION

// ---- VISUs/Visu pour match/V_Match.TcVIS
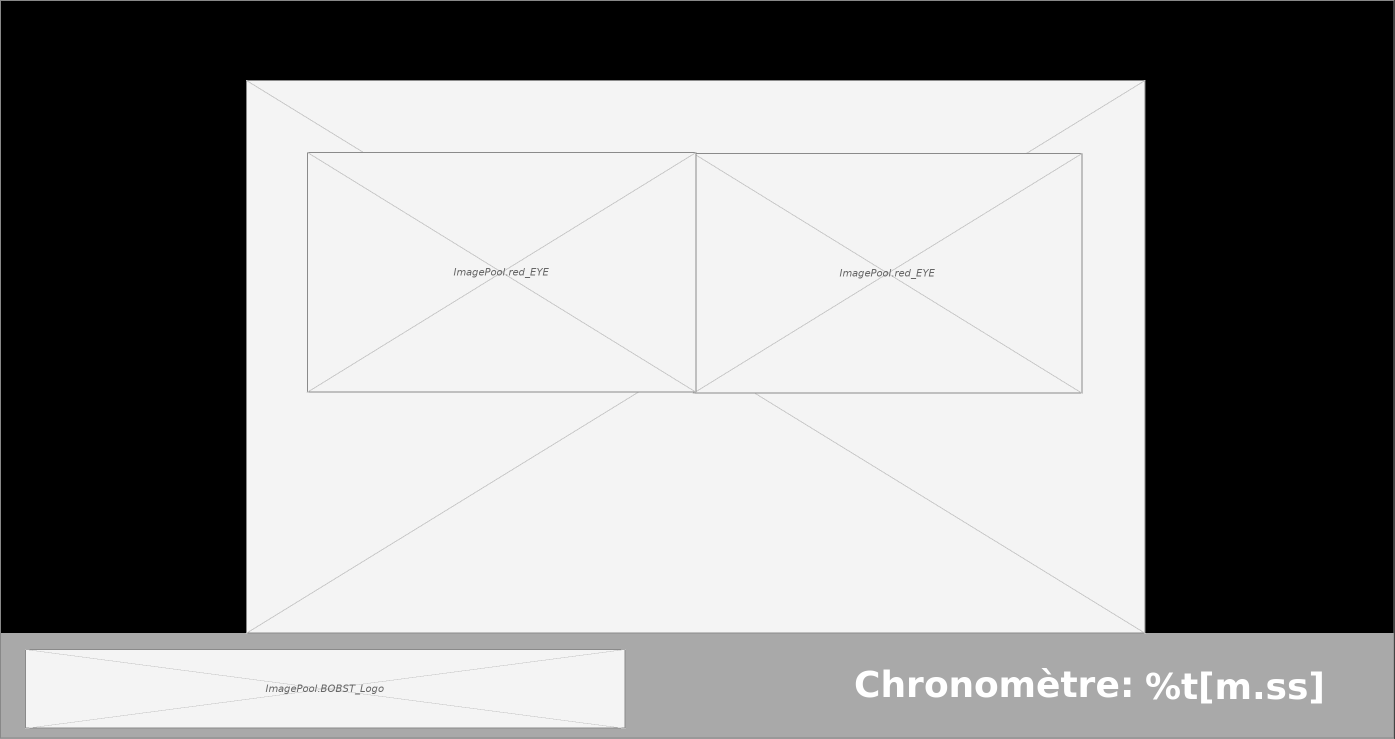
VISUALIZATION V_Match  // 1395x739
    Rectangle (-2,633 1396x109)
    Group (851,647 541x77)
        Label (0,0 400x75), "Chronomètre:"
        Textfield (291,2 250x75), "%t[m.ss]", text variable: G_Match.TimeMatch
    Image (25,649 600x79), image: ImagePool.BOBST_Logo
        OnMouseDown: change screen: V_Menu
    Image (246,80 899x553), image: ImagePool.EYE
    Image (693,153 389x240), invisible if: Not G_Visus.bMatchEnemi, image: ImagePool.red_EYE
    Image (307,152 389x240), invisible if: Not G_Visus.bMatchEnemi, image: ImagePool.red_EYE
END_VISUALIZATION

// ---- VISUs/V_Menu.TcVIS
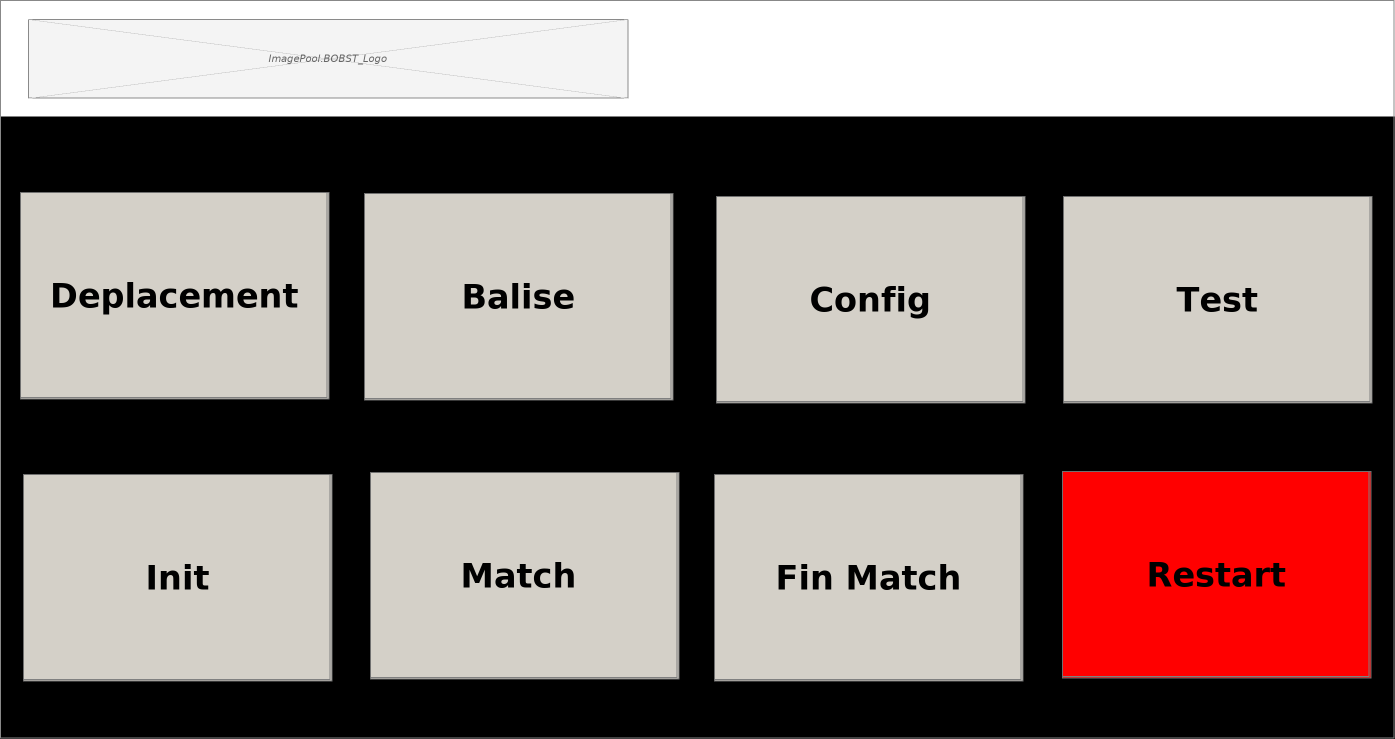
VISUALIZATION V_Menu  // 1395x739
    Rectangle (0,0 1396x116)
    Button (20,192 309x207), "Deplacement"
        OnMouseClick: change screen: V_Deplacement
    Image (28,19 600x79), image: ImagePool.BOBST_Logo
    Button (364,193 309x207), "Balise"
        OnMouseClick: change screen: V_Balise
    Button (716,196 309x207), "Config"
        OnMouseClick: change screen: V_Config
    Button (370,472 309x207), "Match"
        OnMouseClick: change screen: V_Match
    Button (23,474 309x207), "Init"
        OnMouseClick: change screen: V_Init
    Button (714,474 309x207), "Fin Match"
        OnMouseClick: change screen: V_Fin_Match
    Button (1063,196 309x207), "Test"
        OnMouseClick: change screen: V_Test
    Button (1062,471 309x207), "Restart"
        OnMouseClick: toggle G_Visus.bMenuRestart
END_VISUALIZATION
